   W_o[8,37] := -0.1157986;
   W_o[8,38] := 0.2580299;
   W_o[8,39] := 0.220136;
   W_o[9,0] := -0.3132641;
   W_o[9,1] := -0.06183321;
   W_o[9,2] := -0.1190897;
   W_o[9,3] := -0.1472712;
   W_o[9,4] := -0.2051323;
   W_o[9,5] := -0.619219;
   W_o[9,6] := 0.1387524;
   W_o[9,7] := -0.3166307;
   W_o[9,8] := -0.9589977;
   W_o[9,9] := 0.0739672;
   W_o[9,10] := -0.3332131;
   W_o[9,11] := 0.07539017;
   W_o[9,12] := 0.04058671;
   W_o[9,13] := -0.03272064;
   W_o[9,14] := 0.00082348;
   W_o[9,15] := 0.03252422;
   W_o[9,16] := -0.187089;
   W_o[9,17] := 0.03206202;
   W_o[9,18] := -0.1109974;
   W_o[9,19] := -0.2095204;
   W_o[9,20] := -0.5135113;
   W_o[9,21] := 0.1920649;
   W_o[9,22] := -0.01424127;
   W_o[9,23] := -0.00173319;
   W_o[9,24] := -0.08532184;
   W_o[9,25] := -0.2821319;
   W_o[9,26] := -0.03178848;
   W_o[9,27] := -0.0577799;
   W_o[9,28] := 0.2315015;
   W_o[9,29] := 0.07085361;
   W_o[9,30] := 0.1951047;
   W_o[9,31] := 0.08876722;
   W_o[9,32] := 0.1402373;
   W_o[9,33] := 0.2821989;
   W_o[9,34] := 0.1606525;
   W_o[9,35] := -0.1928923;
   W_o[9,36] := 0.01568728;
   W_o[9,37] := -0.1860046;
   W_o[9,38] := 0.09268271;
   W_o[9,39] := -0.01587286;
   W_o[10,0] := -0.02192705;
   W_o[10,1] := 0.2329542;
   W_o[10,2] := -0.00188665;
   W_o[10,3] := 0.143792;
   W_o[10,4] := 0.2532279;
   W_o[10,5] := 0.4542165;
   W_o[10,6] := 0.3260326;
   W_o[10,7] := 0.1298785;
   W_o[10,8] := -0.03717055;
   W_o[10,9] := 0.06002445;
   W_o[10,10] := -0.01521991;
   W_o[10,11] := -0.3110218;
   W_o[10,12] := -0.2009706;
   W_o[10,13] := 0.05733368;
   W_o[10,14] := -0.3404011;
   W_o[10,15] := -0.4737233;
   W_o[10,16] := 0.03586001;
   W_o[10,17] := 0.122371;
   W_o[10,18] := 0.3001329;
   W_o[10,19] := -0.05952299;
   W_o[10,20] := -0.1222852;
   W_o[10,21] := 0.1644575;
   W_o[10,22] := 0.350365;
   W_o[10,23] := -0.3212706;
   W_o[10,24] := 1.075127;
   W_o[10,25] := 1.031375;
   W_o[10,26] := -0.0865766;
   W_o[10,27] := -0.3474564;
   W_o[10,28] := 0.09863426;
   W_o[10,29] := -0.2132783;
   W_o[10,30] := 0.3851247;
   W_o[10,31] := 0.1182251;
   W_o[10,32] := 0.3440039;
   W_o[10,33] := 0.3899197;
   W_o[10,34] := 0.7392653;
   W_o[10,35] := 0.2004149;
   W_o[10,36] := -0.05608039;
   W_o[10,37] := 0.2275992;
   W_o[10,38] := -0.04267087;
   W_o[10,39] := 0.2836826;
   W_o[11,0] := -0.1809653;
   W_o[11,1] := 0.1015071;
   W_o[11,2] := -0.1359787;
   W_o[11,3] := -0.339222;
   W_o[11,4] := 0.01738593;
   W_o[11,5] := 0.00192241;
   W_o[11,6] := -0.02194121;
   W_o[11,7] := -0.1547077;
   W_o[11,8] := 0.06660517;
   W_o[11,9] := -0.1348383;
   W_o[11,10] := -0.134767;
   W_o[11,11] := -0.1782693;
   W_o[11,12] := 0.1472701;
   W_o[11,13] := -0.2786617;
   W_o[11,14] := 0.09056337;
   W_o[11,15] := -0.07600223;
   W_o[11,16] := 0.0426885;
   W_o[11,17] := 0.1939706;
   W_o[11,18] := 0.06352299;
   W_o[11,19] := -0.3184692;
   W_o[11,20] := -0.08175273;
   W_o[11,21] := 0.156256;
   W_o[11,22] := -0.1318633;
   W_o[11,23] := -0.4227056;
   W_o[11,24] := 0.03163491;
   W_o[11,25] := 0.3073466;
   W_o[11,26] := 0.1847536;
   W_o[11,27] := -0.1969137;
   W_o[11,28] := 0.1285785;
   W_o[11,29] := 0.02137278;
   W_o[11,30] := -0.08936202;
   W_o[11,31] := 0.2781714;
   W_o[11,32] := -0.09503862;
   W_o[11,33] := -0.1658657;
   W_o[11,34] := -0.1278383;
   W_o[11,35] := -0.1624458;
   W_o[11,36] := 0.1902921;
   W_o[11,37] := 0.127865;
   W_o[11,38] := -0.07075812;
   W_o[11,39] := 0.428382;
   W_o[12,0] := -0.1219991;
   W_o[12,1] := 0.03823468;
   W_o[12,2] := 0.01577434;
   W_o[12,3] := 0.1470047;
   W_o[12,4] := 0.0760267;
   W_o[12,5] := -0.05943288;
   W_o[12,6] := 0.1218424;
   W_o[12,7] := -0.4092018;
   W_o[12,8] := -0.01477545;
   W_o[12,9] := 0.1050386;
   W_o[12,10] := -0.06524223;
   W_o[12,11] := -0.04999274;
   W_o[12,12] := 0.3521778;
   W_o[12,13] := -0.07877419;
   W_o[12,14] := 0.09900068;
   W_o[12,15] := 0.05063246;
   W_o[12,16] := 0.1021576;
   W_o[12,17] := -0.1172289;
   W_o[12,18] := 0.0756586;
   W_o[12,19] := -0.08223618;
   W_o[12,20] := -0.2851469;
   W_o[12,21] := -0.00324072;
   W_o[12,22] := 0.0636245;
   W_o[12,23] := -0.1829358;
   W_o[12,24] := -0.3075816;
   W_o[12,25] := -0.2720142;
   W_o[12,26] := 0.1688922;
   W_o[12,27] := 0.06790268;
   W_o[12,28] := 0.09229479;
   W_o[12,29] := -0.02702256;
   W_o[12,30] := 0.04384379;
   W_o[12,31] := -0.2710299;
   W_o[12,32] := -0.1930007;
   W_o[12,33] := 0.3236164;
   W_o[12,34] := 0.00694379;
   W_o[12,35] := 0.05657077;
   W_o[12,36] := -0.1271545;
   W_o[12,37] := -0.1242922;
   W_o[12,38] := 0.2896774;
   W_o[12,39] := -0.08116662;
   W_o[13,0] := 0.368947;
   W_o[13,1] := 0.1130772;
   W_o[13,2] := 0.5471025;
   W_o[13,3] := -0.3829838;
   W_o[13,4] := 0.6498483;
   W_o[13,5] := -0.2602773;
   W_o[13,6] := 0.2094651;
   W_o[13,7] := 0.02607361;
   W_o[13,8] := -0.1112638;
   W_o[13,9] := -0.06411502;
   W_o[13,10] := -0.03624791;
   W_o[13,11] := -0.04085876;
   W_o[13,12] := -0.3497492;
   W_o[13,13] := -0.1605573;
   W_o[13,14] := 0.1782783;
   W_o[13,15] := -0.04494572;
   W_o[13,16] := 0.1499656;
   W_o[13,17] := -0.1109314;
   W_o[13,18] := 0.5331051;
   W_o[13,19] := -0.4442391;
   W_o[13,20] := -0.07231531;
   W_o[13,21] := 0.3642985;
   W_o[13,22] := 0.5776525;
   W_o[13,23] := -0.1446741;
   W_o[13,24] := 1.537843;
   W_o[13,25] := 1.406464;
   W_o[13,26] := -0.1982083;
   W_o[13,27] := 0.2525975;
   W_o[13,28] := 0.1090571;
   W_o[13,29] := -0.3863609;
   W_o[13,30] := 0.3198679;
   W_o[13,31] := -0.0655776;
   W_o[13,32] := 0.1591396;
   W_o[13,33] := 0.3302372;
   W_o[13,34] := 0.8010866;
   W_o[13,35] := 0.00219575;
   W_o[13,36] := 0.3194016;
   W_o[13,37] := 0.3292364;
   W_o[13,38] := 0.2895371;
   W_o[13,39] := 0.1438104;
   W_o[14,0] := -0.06043304;
   W_o[14,1] := 0.1463838;
   W_o[14,2] := 0.1813115;
   W_o[14,3] := -0.4461174;
   W_o[14,4] := -0.08022243;
   W_o[14,5] := 0.1215249;
   W_o[14,6] := -0.09096271;
   W_o[14,7] := -0.08817829;
   W_o[14,8] := -0.4104892;
   W_o[14,9] := 0.00550563;
   W_o[14,10] := 0.02338252;
   W_o[14,11] := 0.03576816;
   W_o[14,12] := 0.09025624;
   W_o[14,13] := -0.165952;
   W_o[14,14] := -0.1859627;
   W_o[14,15] := -0.09394215;
   W_o[14,16] := -0.06208068;
   W_o[14,17] := -0.00717838;
   W_o[14,18] := 0.1996924;
   W_o[14,19] := 0.01073706;
   W_o[14,20] := -0.1823136;
   W_o[14,21] := 0.01420894;
   W_o[14,22] := -0.1017454;
   W_o[14,23] := -0.4975724;
   W_o[14,24] := -0.4672968;
   W_o[14,25] := -0.2924049;
   W_o[14,26] := -0.190528;
   W_o[14,27] := -0.1670942;
   W_o[14,28] := -0.01935058;
   W_o[14,29] := -0.1424983;
   W_o[14,30] := -0.1588129;
   W_o[14,31] := 0.2039351;
   W_o[14,32] := -0.06176985;
   W_o[14,33] := 0.1746421;
   W_o[14,34] := 0.2394749;
   W_o[14,35] := -0.1960727;
   W_o[14,36] := 0.05518134;
   W_o[14,37] := 0.09389904;
   W_o[14,38] := 0.08116579;
   W_o[14,39] := 0.1385406;
   W_o[15,0] := -0.2035415;
   W_o[15,1] := 0.2229884;
   W_o[15,2] := -0.7284631;
   W_o[15,3] := 0.1279051;
   W_o[15,4] := -0.000869;
   W_o[15,5] := 0.5366808;
   W_o[15,6] := -0.01224643;
   W_o[15,7] := 0.1336179;
   W_o[15,8] := -0.3520414;
   W_o[15,9] := -0.00480295;
   W_o[15,10] := 0.1333943;
   W_o[15,11] := 0.05102095;
   W_o[15,12] := -0.05708028;
   W_o[15,13] := -0.06014942;
   W_o[15,14] := 0.01049514;
   W_o[15,15] := -0.09353844;
   W_o[15,16] := 0.07731096;
   W_o[15,17] := 0.01013883;
   W_o[15,18] := 0.07310723;
   W_o[15,19] := -0.8692668;
   W_o[15,20] := -0.2155429;
   W_o[15,21] := 0.09906635;
   W_o[15,22] := -0.0306251;
   W_o[15,23] := 0.3455428;
   W_o[15,24] := -0.1861183;
   W_o[15,25] := -0.2109679;
   W_o[15,26] := -0.05899647;
   W_o[15,27] := 0.01260784;
   W_o[15,28] := 0.04030582;
   W_o[15,29] := 0.1423471;
   W_o[15,30] := 0.2868683;
   W_o[15,31] := 0.1026989;
   W_o[15,32] := 0.2412259;
   W_o[15,33] := -0.04419544;
   W_o[15,34] := 0.1289678;
   W_o[15,35] := -0.2943439;
   W_o[15,36] := -0.00652304;
   W_o[15,37] := -0.03412445;
   W_o[15,38] := 0.4802624;
   W_o[15,39] := 0.2227584;
   R_i[0,0] := -0.01601154;
   R_i[0,1] := -0.4505664;
   R_i[0,2] := 0.3115061;
   R_i[0,3] := 0.7538006;
   R_i[0,4] := -0.1402078;
   R_i[0,5] := -0.04954997;
   R_i[0,6] := -0.08327835;
   R_i[0,7] := 0.3733349;
   R_i[0,8] := 0.6963265;
   R_i[0,9] := 0.2863626;
   R_i[0,10] := 0.7997712;
   R_i[0,11] := -0.7498176;
   R_i[0,12] := -0.6526057;
   R_i[0,13] := 0.1387625;
   R_i[0,14] := 0.08631746;
   R_i[0,15] := 0.05898035;
   R_i[1,0] := -0.401232;
   R_i[1,1] := 0.7335209;
   R_i[1,2] := -0.09579885;
   R_i[1,3] := 0.02985846;
   R_i[1,4] := -0.3186485;
   R_i[1,5] := -0.2394537;
   R_i[1,6] := 0.5418519;
   R_i[1,7] := -0.2710277;
   R_i[1,8] := 0.00622073;
   R_i[1,9] := 0.09155256;
   R_i[1,10] := 0.1461604;
   R_i[1,11] := -0.0016893;
   R_i[1,12] := 0.2237979;
   R_i[1,13] := 0.1673195;
   R_i[1,14] := -0.07847317;
   R_i[1,15] := -0.07302959;
   R_i[2,0] := 0.2143267;
   R_i[2,1] := -0.5247285;
   R_i[2,2] := 0.3322655;
   R_i[2,3] := 0.2965375;
   R_i[2,4] := 0.1318167;
   R_i[2,5] := 0.1446274;
   R_i[2,6] := -0.130442;
   R_i[2,7] := -0.1195364;
   R_i[2,8] := -0.3126507;
   R_i[2,9] := -0.240243;
   R_i[2,10] := 0.08897854;
   R_i[2,11] := -0.3383393;
   R_i[2,12] := -0.1979901;
   R_i[2,13] := 0.07993159;
   R_i[2,14] := -0.1129293;
   R_i[2,15] := -0.07898453;
   R_i[3,0] := 0.2161791;
   R_i[3,1] := 0.14047;
   R_i[3,2] := -0.339711;
   R_i[3,3] := -0.8781343;
   R_i[3,4] := 0.1890773;
   R_i[3,5] := -0.08525109;
   R_i[3,6] := 0.00524858;
   R_i[3,7] := 0.6169428;
   R_i[3,8] := -0.02290213;
   R_i[3,9] := -0.1232494;
   R_i[3,10] := 0.1836437;
   R_i[3,11] := -0.0097614;
   R_i[3,12] := -0.00912099;
   R_i[3,13] := 0.08642489;
   R_i[3,14] := -0.1198076;
   R_i[3,15] := -0.1218542;
   R_i[4,0] := -0.1688442;
   R_i[4,1] := -0.01549527;
   R_i[4,2] := -0.09087992;
   R_i[4,3] := 0.2035424;
   R_i[4,4] := 0.03523245;
   R_i[4,5] := -0.7966576;
   R_i[4,6] := 0.01135984;
   R_i[4,7] := 0.1643567;
   R_i[4,8] := 0.2464019;
   R_i[4,9] := 0.348982;
   R_i[4,10] := 0.1028246;
   R_i[4,11] := 0.00752686;
   R_i[4,12] := 0.04740289;
   R_i[4,13] := 0.6564606;
   R_i[4,14] := 0.3415406;
   R_i[4,15] := -0.1820581;
   R_i[5,0] := 0.14134;
   R_i[5,1] := -0.5241947;
   R_i[5,2] := 0.2979371;
   R_i[5,3] := 0.5492764;
   R_i[5,4] := -0.5426098;
   R_i[5,5] := -0.5120263;
   R_i[5,6] := -0.6021063;
   R_i[5,7] := -0.5658756;
   R_i[5,8] := 0.2832164;
   R_i[5,9] := 0.2791682;
   R_i[5,10] := 0.0495842;
   R_i[5,11] := -0.4578474;
   R_i[5,12] := -0.6485385;
   R_i[5,13] := 0.06905902;
   R_i[5,14] := -0.4043413;
   R_i[5,15] := -0.3203804;
   R_i[6,0] := -0.1409825;
   R_i[6,1] := -0.5848475;
   R_i[6,2] := 0.1453531;
   R_i[6,3] := 0.07121052;
   R_i[6,4] := -0.3604121;
   R_i[6,5] := -0.397943;
   R_i[6,6] := -1.122013;
   R_i[6,7] := -0.1309183;
   R_i[6,8] := -0.191392;
   R_i[6,9] := 0.02611434;
   R_i[6,10] := -0.2210553;
   R_i[6,11] := 0.03291342;
   R_i[6,12] := -0.3278158;
   R_i[6,13] := 0.3461519;
   R_i[6,14] := 0.2672345;
   R_i[6,15] := 0.1619738;
   R_i[7,0] := -0.1475523;
   R_i[7,1] := -0.6828271;
   R_i[7,2] := -0.2710959;
   R_i[7,3] := 0.3215815;
   R_i[7,4] := 0.03019373;
   R_i[7,5] := 0.1696624;
   R_i[7,6] := 0.1198417;
   R_i[7,7] := -0.1019654;
   R_i[7,8] := 0.5909069;
   R_i[7,9] := -0.3902815;
   R_i[7,10] := 0.2400998;
   R_i[7,11] := -0.3905518;
   R_i[7,12] := -0.3868088;
   R_i[7,13] := -0.1764367;
   R_i[7,14] := 0.2387517;
   R_i[7,15] := -0.1071883;
   R_i[8,0] := -0.23345;
   R_i[8,1] := -0.3877599;
   R_i[8,2] := -0.3317247;
   R_i[8,3] := 0.1490105;
   R_i[8,4] := 0.07190004;
   R_i[8,5] := -0.05165868;
   R_i[8,6] := 0.4919274;
   R_i[8,7] := 0.6358661;
   R_i[8,8] := -0.1297378;
   R_i[8,9] := -0.3915481;
   R_i[8,10] := 0.01818666;
   R_i[8,11] := -0.3103262;
   R_i[8,12] := -0.2901289;
   R_i[8,13] := -0.01039465;
   R_i[8,14] := 0.194509;
   R_i[8,15] := -0.2007908;
   R_i[9,0] := -0.2780712;
   R_i[9,1] := 0.00795646;
   R_i[9,2] := 0.1596926;
   R_i[9,3] := -0.09819215;
   R_i[9,4] := 0.00536336;
   R_i[9,5] := -0.01222592;
   R_i[9,6] := 0.05426886;
   R_i[9,7] := -0.2209529;
   R_i[9,8] := 0.1505673;
   R_i[9,9] := -0.2607254;
   R_i[9,10] := 0.3316929;
   R_i[9,11] := 0.1011708;
   R_i[9,12] := -0.2139317;
   R_i[9,13] := 0.4217584;
   R_i[9,14] := 0.01216281;
   R_i[9,15] := -0.0816205;
   R_i[10,0] := 0.126458;
   R_i[10,1] := 0.02421534;
   R_i[10,2] := -0.2489259;
   R_i[10,3] := 0.09164374;
   R_i[10,4] := -0.4294859;
   R_i[10,5] := -0.0543494;
   R_i[10,6] := 0.5646753;
   R_i[10,7] := 0.331787;
   R_i[10,8] := 0.2602156;
   R_i[10,9] := -0.3929808;
   R_i[10,10] := -0.395796;
   R_i[10,11] := -0.00741246;
   R_i[10,12] := -0.3358352;
   R_i[10,13] := -0.0185852;
   R_i[10,14] := 0.4410301;
   R_i[10,15] := -0.09651927;
   R_i[11,0] := 0.09693456;
   R_i[11,1] := -0.3512501;
   R_i[11,2] := -0.02015482;
   R_i[11,3] := 0.3572097;
   R_i[11,4] := -0.1196542;
   R_i[11,5] := 0.1445999;
   R_i[11,6] := -0.1906793;
   R_i[11,7] := 0.08080416;
   R_i[11,8] := 0.1779785;
   R_i[11,9] := -0.1425034;
   R_i[11,10] := -0.3862794;
   R_i[11,11] := 0.4956163;
   R_i[11,12] := -0.1790929;
   R_i[11,13] := 0.2083636;
   R_i[11,14] := 0.4006914;
   R_i[11,15] := 0.3896022;
   R_i[12,0] := 0.3400891;
   R_i[12,1] := -0.1727159;
   R_i[12,2] := -0.3076965;
   R_i[12,3] := -0.2823079;
   R_i[12,4] := 0.0525449;
   R_i[12,5] := 0.07448359;
   R_i[12,6] := -0.00981909;
   R_i[12,7] := 0.1008154;
   R_i[12,8] := 0.3009783;
   R_i[12,9] := 0.2912007;
   R_i[12,10] := 0.1271894;
   R_i[12,11] := -0.06783659;
   R_i[12,12] := 0.4455962;
   R_i[12,13] := -0.3242948;
   R_i[12,14] := -0.183432;
   R_i[12,15] := -0.1089303;
   R_i[13,0] := -0.2894851;
   R_i[13,1] := -0.1664966;
   R_i[13,2] := 0.04430598;
   R_i[13,3] := 0.1107857;
   R_i[13,4] := -0.5688026;
   R_i[13,5] := -0.07979194;
   R_i[13,6] := 0.1527517;
   R_i[13,7] := 0.1273375;
   R_i[13,8] := 0.3621153;
   R_i[13,9] := 0.3043333;
   R_i[13,10] := -0.1798581;
   R_i[13,11] := -0.237729;
   R_i[13,12] := 0.1235583;
   R_i[13,13] := 0.5035439;
   R_i[13,14] := 0.108624;
   R_i[13,15] := -0.02580172;
   R_i[14,0] := 0.04543614;
   R_i[14,1] := -0.4043088;
   R_i[14,2] := 0.1209751;
   R_i[14,3] := 0.4883763;
   R_i[14,4] := 0.00980398;
   R_i[14,5] := 0.03799421;
   R_i[14,6] := 0.3278515;
   R_i[14,7] := 0.0660439;
   R_i[14,8] := 0.172085;
   R_i[14,9] := -0.3707425;
   R_i[14,10] := -0.1385914;
   R_i[14,11] := 0.2718971;
   R_i[14,12] := -0.1328888;
   R_i[14,13] := 0.2701875;
   R_i[14,14] := 1.386678;
   R_i[14,15] := 0.05095792;
   R_i[15,0] := 0.1214196;
   R_i[15,1] := -0.03100028;
   R_i[15,2] := 0.2684634;
   R_i[15,3] := 0.2103243;
   R_i[15,4] := -0.1190422;
   R_i[15,5] := 0.09452529;
   R_i[15,6] := 0.3082354;
   R_i[15,7] := -3.856E-05;
   R_i[15,8] := 0.2727255;
   R_i[15,9] := 0.05441154;
   R_i[15,10] := -0.1230815;
   R_i[15,11] := -0.4781843;
   R_i[15,12] := -0.2143165;
   R_i[15,13] := -0.2471516;
   R_i[15,14] := 0.2087188;
   R_i[15,15] := 0.02325043;
   R_f[0,0] := -0.03493118;
   R_f[0,1] := -0.3783333;
   R_f[0,2] := 0.03728793;
   R_f[0,3] := 0.1427855;
   R_f[0,4] := -0.1200396;
   R_f[0,5] := -0.06856227;
   R_f[0,6] := 0.07930882;
   R_f[0,7] := 0.2776607;
   R_f[0,8] := 0.07494716;
   R_f[0,9] := 0.1461581;
   R_f[0,10] := -0.07652009;
   R_f[0,11] := -0.09052465;
   R_f[0,12] := -0.1157662;
   R_f[0,13] := 0.04987612;
   R_f[0,14] := 0.06529343;
   R_f[0,15] := 0.00263772;
   R_f[1,0] := -0.4377774;
   R_f[1,1] := 0.7251403;
   R_f[1,2] := -0.3877139;
   R_f[1,3] := -0.0144369;
   R_f[1,4] := -0.00149874;
   R_f[1,5] := -0.3447672;
   R_f[1,6] := 0.2917376;
   R_f[1,7] := 0.09541123;
   R_f[1,8] := 0.3457976;
   R_f[1,9] := 0.6298571;
   R_f[1,10] := 0.05302448;
   R_f[1,11] := 0.2072578;
   R_f[1,12] := -0.04234733;
   R_f[1,13] := 0.3336825;
   R_f[1,14] := 0.1307107;
   R_f[1,15] := 0.1257179;
   R_f[2,0] := 0.3310767;
   R_f[2,1] := -0.3810703;
   R_f[2,2] := 0.1153975;
   R_f[2,3] := 0.3476575;
   R_f[2,4] := -0.2480675;
   R_f[2,5] := 0.1239669;
   R_f[2,6] := -0.0001569;
   R_f[2,7] := -0.03111286;
   R_f[2,8] := -0.4061953;
   R_f[2,9] := -0.1027613;
   R_f[2,10] := -0.01848604;
   R_f[2,11] := -0.3815011;
   R_f[2,12] := 0.07561549;
   R_f[2,13] := -0.3294232;
   R_f[2,14] := -0.04146929;
   R_f[2,15] := 0.1021808;
   R_f[3,0] := -0.9564785;
   R_f[3,1] := 0.3263851;
   R_f[3,2] := -0.1824219;
   R_f[3,3] := -0.2994925;
   R_f[3,4] := 0.1714023;
   R_f[3,5] := -0.2092119;
   R_f[3,6] := -0.1032977;
   R_f[3,7] := -0.1582146;
   R_f[3,8] := 0.1507048;
   R_f[3,9] := 0.337986;
   R_f[3,10] := -0.2794919;
   R_f[3,11] := 0.08474356;
   R_f[3,12] := 0.2481105;
   R_f[3,13] := 0.09939278;
   R_f[3,14] := -0.2410131;
   R_f[3,15] := -0.1935376;
   R_f[4,0] := -0.234988;
   R_f[4,1] := -0.4074499;
   R_f[4,2] := 0.2635157;
   R_f[4,3] := -0.2668453;
   R_f[4,4] := -0.09082807;
   R_f[4,5] := -0.08405253;
   R_f[4,6] := 0.08696185;
   R_f[4,7] := 0.1112983;
   R_f[4,8] := 0.1638763;
   R_f[4,9] := -0.1186807;
   R_f[4,10] := 0.3262174;
   R_f[4,11] := -0.1426349;
   R_f[4,12] := 0.1308399;
   R_f[4,13] := 0.1795556;
   R_f[4,14] := 0.1659483;
   R_f[4,15] := 0.1235942;
   R_f[5,0] := 0.3548082;
   R_f[5,1] := -0.1270981;
   R_f[5,2] := 0.2426847;
   R_f[5,3] := 0.0801195;
   R_f[5,4] := 0.2115624;
   R_f[5,5] := 0.2757975;
   R_f[5,6] := 0.2001711;
   R_f[5,7] := 0.01883883;
   R_f[5,8] := -0.3942798;
   R_f[5,9] := -0.3586779;
   R_f[5,10] := 0.06389395;
   R_f[5,11] := -0.1110686;
   R_f[5,12] := 0.1175703;
   R_f[5,13] := -0.0187532;
   R_f[5,14] := 0.01303833;
   R_f[5,15] := -0.0669001;
   R_f[6,0] := -0.5004723;
   R_f[6,1] := -0.07684148;
   R_f[6,2] := 0.1981799;
   R_f[6,3] := 0.0597102;
   R_f[6,4] := -0.04680483;
   R_f[6,5] := 0.317703;
   R_f[6,6] := 0.1253361;
   R_f[6,7] := 0.1381588;
   R_f[6,8] := 0.02148284;
   R_f[6,9] := -0.0610669;
   R_f[6,10] := 0.1336211;
   R_f[6,11] := 0.2163607;
   R_f[6,12] := -0.09828766;
   R_f[6,13] := 0.2164403;
   R_f[6,14] := 0.2033899;
   R_f[6,15] := 0.1417818;
   R_f[7,0] := 0.2612512;
   R_f[7,1] := -0.03714739;
   R_f[7,2] := 0.08117681;
   R_f[7,3] := 0.20745;
   R_f[7,4] := -0.320446;
   R_f[7,5] := 0.4126448;
   R_f[7,6] := 0.616157;
   R_f[7,7] := -0.1764756;
   R_f[7,8] := -0.1566713;
   R_f[7,9] := -0.02732511;
   R_f[7,10] := -0.4989151;
   R_f[7,11] := 0.00061774;
   R_f[7,12] := -0.02982556;
   R_f[7,13] := 0.03914607;
   R_f[7,14] := 0.2035217;
   R_f[7,15] := 0.01521025;
   R_f[8,0] := -0.00262567;
   R_f[8,1] := -0.1957263;
   R_f[8,2] := -0.0133352;
   R_f[8,3] := 0.1326498;
   R_f[8,4] := -0.06475109;
   R_f[8,5] := 0.2750055;
   R_f[8,6] := 0.2935895;
   R_f[8,7] := 0.1078199;
   R_f[8,8] := -0.5541819;
   R_f[8,9] := -0.03762578;
   R_f[8,10] := -0.2519385;
   R_f[8,11] := 0.277219;
   R_f[8,12] := -0.1539617;
   R_f[8,13] := -0.02145483;
   R_f[8,14] := 0.2416782;
   R_f[8,15] := 0.06824671;
   R_f[9,0] := 0.2504059;
   R_f[9,1] := -0.3383861;
   R_f[9,2] := 0.0674123;
   R_f[9,3] := 0.2097046;
   R_f[9,4] := -0.0898691;
   R_f[9,5] := -0.2091327;
   R_f[9,6] := 0.3162811;
   R_f[9,7] := 0.265341;
   R_f[9,8] := 0.02326944;
   R_f[9,9] := -0.8053678;
   R_f[9,10] := -0.2416072;
   R_f[9,11] := -0.03336972;
   R_f[9,12] := -0.3634549;
   R_f[9,13] := 0.01661946;
   R_f[9,14] := -0.117901;
   R_f[9,15] := 0.1400468;
   R_f[10,0] := 0.2025216;
   R_f[10,1] := -0.3309455;
   R_f[10,2] := 0.2834905;
   R_f[10,3] := 0.2098317;
   R_f[10,4] := -0.3916658;
   R_f[10,5] := 0.1489443;
   R_f[10,6] := 0.05038162;
   R_f[10,7] := 0.1421797;
   R_f[10,8] := -0.2475107;
   R_f[10,9] := 0.04759743;
   R_f[10,10] := -0.1642638;
   R_f[10,11] := -0.1621708;
   R_f[10,12] := -0.1235068;
   R_f[10,13] := 0.08995254;
   R_f[10,14] := -0.01327613;
   R_f[10,15] := 0.2285491;
   R_f[11,0] := 0.1601221;
   R_f[11,1] := 0.2628818;
   R_f[11,2] := 0.2190603;
   R_f[11,3] := -0.04701964;
   R_f[11,4] := -0.1388493;
   R_f[11,5] := 0.08709867;
   R_f[11,6] := -0.07009537;
   R_f[11,7] := -0.1695109;
   R_f[11,8] := 0.02868164;
   R_f[11,9] := -0.0112115;
   R_f[11,10] := 0.07267684;
   R_f[11,11] := -0.1989551;
   R_f[11,12] := 0.3613658;
   R_f[11,13] := -0.05935945;
   R_f[11,14] := 0.0822355;
   R_f[11,15] := 0.373795;
   R_f[12,0] := -0.2599636;
   R_f[12,1] := -0.4840415;
   R_f[12,2] := -0.3295081;
   R_f[12,3] := 0.1110019;
   R_f[12,4] := -0.2677098;
   R_f[12,5] := -0.1735305;
   R_f[12,6] := 0.1697096;
   R_f[12,7] := -0.3476382;
   R_f[12,8] := 0.517248;
   R_f[12,9] := -0.2285556;
   R_f[12,10] := 0.86062;
   R_f[12,11] := 0.06095523;
   R_f[12,12] := -0.1267713;
   R_f[12,13] := 0.2335584;
   R_f[12,14] := 0.2402046;
   R_f[12,15] := -0.2279788;
   R_f[13,0] := 0.02567713;
   R_f[13,1] := -0.3151536;
   R_f[13,2] := -0.1262183;
   R_f[13,3] := 0.1836853;
   R_f[13,4] := -0.03905401;
   R_f[13,5] := 0.7135632;
   R_f[13,6] := 0.08130559;
   R_f[13,7] := 0.01576971;
   R_f[13,8] := -0.2050417;
   R_f[13,9] := 0.07079811;
   R_f[13,10] := -0.1090281;
   R_f[13,11] := 0.1574726;
   R_f[13,12] := -0.3404612;
   R_f[13,13] := 0.1042019;
   R_f[13,14] := -0.05406023;
   R_f[13,15] := 0.2302613;
   R_f[14,0] := 0.05553682;
   R_f[14,1] := 0.03039004;
   R_f[14,2] := -0.3977577;
   R_f[14,3] := 0.1773666;
   R_f[14,4] := -0.1401487;
   R_f[14,5] := 0.1813615;
   R_f[14,6] := 0.08784663;
   R_f[14,7] := -0.00406716;
   R_f[14,8] := 0.2937247;
   R_f[14,9] := -0.2185726;
   R_f[14,10] := 0.3286898;
   R_f[14,11] := 0.5202897;
   R_f[14,12] := 0.2797473;
   R_f[14,13] := -0.109547;
   R_f[14,14] := 1.174732;
   R_f[14,15] := 0.2927172;
   R_f[15,0] := 0.3542146;
   R_f[15,1] := -0.6242056;
   R_f[15,2] := 0.2294325;
   R_f[15,3] := 0.2983122;
   R_f[15,4] := -0.2018091;
   R_f[15,5] := 0.3988208;
   R_f[15,6] := 0.2762798;
   R_f[15,7] := 0.3846879;
   R_f[15,8] := 0.04349254;
   R_f[15,9] := -0.1081066;
   R_f[15,10] := -0.3734537;
   R_f[15,11] := -0.1098458;
   R_f[15,12] := 0.3364737;
   R_f[15,13] := 0.3455147;
   R_f[15,14] := 0.02944022;
   R_f[15,15] := 0.02307001;
   R_g[0,0] := -1.251124;
   R_g[0,1] := -0.2188334;
   R_g[0,2] := 0.1101293;
   R_g[0,3] := 0.2501267;
   R_g[0,4] := -0.1040586;
   R_g[0,5] := 0.1389121;
   R_g[0,6] := 0.1024126;
   R_g[0,7] := 0.2224759;
   R_g[0,8] := 0.06886309;
   R_g[0,9] := -0.05504098;
   R_g[0,10] := 0.1316268;
   R_g[0,11] := -0.09226879;
   R_g[0,12] := 0.03665201;
   R_g[0,13] := 0.01448225;
   R_g[0,14] := 0.08514914;
   R_g[0,15] := 0.1034982;
   R_g[1,0] := -0.01289242;
   R_g[1,1] := -0.7693796;
   R_g[1,2] := -0.00765862;
   R_g[1,3] := -0.02182954;
   R_g[1,4] := -0.0062479;
   R_g[1,5] := -0.09856889;
   R_g[1,6] := -0.00179921;
   R_g[1,7] := -0.1597593;
   R_g[1,8] := 0.1441042;
   R_g[1,9] := -0.136594;
   R_g[1,10] := -0.1046183;
   R_g[1,11] := 0.1787898;
   R_g[1,12] := 0.1371266;
   R_g[1,13] := 0.1039945;
   R_g[1,14] := 0.2064357;
   R_g[1,15] := 0.05955669;
   R_g[2,0] := -0.00450423;
   R_g[2,1] := 0.2783746;
   R_g[2,2] := -1.652401;
   R_g[2,3] := -0.08348246;
   R_g[2,4] := 0.00295603;
   R_g[2,5] := -0.1220379;
   R_g[2,6] := -0.01780931;
   R_g[2,7] := 0.08614038;
   R_g[2,8] := -0.05562058;
   R_g[2,9] := 0.1005678;
   R_g[2,10] := 0.03247114;
   R_g[2,11] := -0.1122308;
   R_g[2,12] := -0.1009854;
   R_g[2,13] := 0.01667355;
   R_g[2,14] := -0.2604633;
   R_g[2,15] := -0.262483;
   R_g[3,0] := -0.03127015;
   R_g[3,1] := 0.2364704;
   R_g[3,2] := -0.2546491;
   R_g[3,3] := -0.9946523;
   R_g[3,4] := -0.00474326;
   R_g[3,5] := 0.0225782;
   R_g[3,6] := -0.1201107;
   R_g[3,7] := -0.3624461;
   R_g[3,8] := 0.1697178;
   R_g[3,9] := 0.1855698;
   R_g[3,10] := 0.1265972;
   R_g[3,11] := -0.07901487;
   R_g[3,12] := -0.08990744;
   R_g[3,13] := 0.1421835;
   R_g[3,14] := -0.143879;
   R_g[3,15] := -0.2938069;
   R_g[4,0] := 0.07746305;
   R_g[4,1] := 0.05525218;
   R_g[4,2] := 0.1861004;
   R_g[4,3] := 0.1101569;
   R_g[4,4] := -1.795932;
   R_g[4,5] := -0.03749003;
   R_g[4,6] := 0.01035422;
   R_g[4,7] := 0.1005974;
   R_g[4,8] := 0.2383393;
   R_g[4,9] := -0.04896057;
   R_g[4,10] := -0.1035081;
   R_g[4,11] := 0.0563738;
   R_g[4,12] := -0.2545002;
   R_g[4,13] := -0.08886177;
   R_g[4,14] := -0.115833;
   R_g[4,15] := 0.4366852;
   R_g[5,0] := -0.1500607;
   R_g[5,1] := 0.1485784;
   R_g[5,2] := 0.09219331;
   R_g[5,3] := 0.2430712;
   R_g[5,4] := 0.02014972;
   R_g[5,5] := -1.739048;
   R_g[5,6] := -0.06327479;
   R_g[5,7] := 0.09475522;
   R_g[5,8] := -0.0571667;
   R_g[5,9] := 0.00648821;
   R_g[5,10] := -0.08605717;
   R_g[5,11] := 0.04396249;
   R_g[5,12] := 0.1986526;
   R_g[5,13] := 0.2101544;
   R_g[5,14] := -0.04510098;
   R_g[5,15] := -0.05707484;
   R_g[6,0] := 0.05463404;
   R_g[6,1] := -0.2467168;
   R_g[6,2] := 0.1494595;
   R_g[6,3] := 0.2778161;
   R_g[6,4] := 0.05857803;
   R_g[6,5] := -0.09827307;
   R_g[6,6] := -1.369555;
   R_g[6,7] := 0.03997089;
   R_g[6,8] := 0.1069783;
   R_g[6,9] := -0.152829;
   R_g[6,10] := -0.1145824;
   R_g[6,11] := 0.2323128;
   R_g[6,12] := 0.06463466;
   R_g[6,13] := -0.04114177;
   R_g[6,14] := 0.01473683;
   R_g[6,15] := 0.09800901;
   R_g[7,0] := 0.03089882;
   R_g[7,1] := -0.1286617;
   R_g[7,2] := -0.1448888;
   R_g[7,3] := 0.08099888;
   R_g[7,4] := -0.01760847;
   R_g[7,5] := 0.123238;
   R_g[7,6] := 0.01051104;
   R_g[7,7] := -1.431484;
   R_g[7,8] := 0.05538348;
   R_g[7,9] := 0.08765257;
   R_g[7,10] := 0.04525751;
   R_g[7,11] := -0.08530193;
   R_g[7,12] := 0.06940229;
   R_g[7,13] := 0.2047146;
   R_g[7,14] := 0.1114375;
   R_g[7,15] := -0.01617558;
   R_g[8,0] := 0.00375073;
   R_g[8,1] := 0.05561948;
   R_g[8,2] := 0.07504495;
   R_g[8,3] := 0.1384679;
   R_g[8,4] := 0.01292397;
   R_g[8,5] := -0.1276252;
   R_g[8,6] := 0.00967023;
   R_g[8,7] := -0.02755805;
   R_g[8,8] := -1.648121;
   R_g[8,9] := 0.1276399;
   R_g[8,10] := 0.1534631;
   R_g[8,11] := -0.01111799;
   R_g[8,12] := 0.1786743;
   R_g[8,13] := -0.1449942;
   R_g[8,14] := -0.04605825;
   R_g[8,15] := 0.04006226;
   R_g[9,0] := 0.07299295;
   R_g[9,1] := -0.1971753;
   R_g[9,2] := -0.09354591;
   R_g[9,3] := 0.114232;
   R_g[9,4] := 0.1877067;
   R_g[9,5] := -0.1877008;
   R_g[9,6] := 0.1763708;
   R_g[9,7] := -0.00016326;
   R_g[9,8] := 0.05343577;
   R_g[9,9] := -1.985819;
   R_g[9,10] := -0.07635771;
   R_g[9,11] := 0.00779606;
   R_g[9,12] := -0.2143648;
   R_g[9,13] := 0.1459147;
   R_g[9,14] := 0.07554781;
   R_g[9,15] := -0.05975449;
   R_g[10,0] := -0.2548342;
   R_g[10,1] := 0.06535473;
   R_g[10,2] := -0.1516876;
   R_g[10,3] := -0.136762;
   R_g[10,4] := 0.1371599;
   R_g[10,5] := -0.04971113;
   R_g[10,6] := -0.04342166;
   R_g[10,7] := 0.1320384;
   R_g[10,8] := -0.05174213;
   R_g[10,9] := 0.172242;
   R_g[10,10] := -1.545853;
   R_g[10,11] := 0.08824725;
   R_g[10,12] := 0.543172;
   R_g[10,13] := -0.00582574;
   R_g[10,14] := -0.1842785;
   R_g[10,15] := -0.08446352;
   R_g[11,0] := -0.01310127;
   R_g[11,1] := 0.354282;
   R_g[11,2] := -0.2256483;
   R_g[11,3] := -0.4770394;
   R_g[11,4] := 0.02761533;
   R_g[11,5] := -0.02962572;
   R_g[11,6] := 0.06179708;
   R_g[11,7] := -0.0153362;
   R_g[11,8] := 0.04956101;
   R_g[11,9] := 0.1562686;
   R_g[11,10] := -0.1213244;
   R_g[11,11] := -0.9070006;
   R_g[11,12] := 0.2075333;
   R_g[11,13] := -0.08345811;
   R_g[11,14] := -0.3010131;
   R_g[11,15] := -0.3438835;
   R_g[12,0] := 0.1546433;
   R_g[12,1] := -0.1955362;
   R_g[12,2] := 0.2216086;
   R_g[12,3] := 0.3276492;
   R_g[12,4] := 0.02648578;
   R_g[12,5] := 0.09656581;
   R_g[12,6] := 0.09269863;
   R_g[12,7] := -0.00748462;
   R_g[12,8] := 0.2384084;
   R_g[12,9] := -0.2226923;
   R_g[12,10] := -0.1432746;
   R_g[12,11] := 0.1678383;
   R_g[12,12] := -1.566237;
   R_g[12,13] := -0.1101629;
   R_g[12,14] := 0.1427753;
   R_g[12,15] := 0.4183835;
   R_g[13,0] := 0.08890279;
   R_g[13,1] := -0.1990502;
   R_g[13,2] := -0.01056181;
   R_g[13,3] := 0.2478623;
   R_g[13,4] := 0.07754356;
   R_g[13,5] := 0.1655405;
   R_g[13,6] := 0.2601499;
   R_g[13,7] := 0.09906179;
   R_g[13,8] := -0.00865919;
   R_g[13,9] := -0.3019298;
   R_g[13,10] := -0.02393581;
   R_g[13,11] := -0.07343359;
   R_g[13,12] := -0.1289207;
   R_g[13,13] := -1.642736;
   R_g[13,14] := 0.06043187;
   R_g[13,15] := 0.1288359;
   R_g[14,0] := -0.09330796;
   R_g[14,1] := 0.1997155;
   R_g[14,2] := -0.1660388;
   R_g[14,3] := -0.2476246;
   R_g[14,4] := -0.245462;
   R_g[14,5] := -0.2337237;
   R_g[14,6] := -0.02659419;
   R_g[14,7] := 0.105768;
   R_g[14,8] := -0.0639934;
   R_g[14,9] := 0.2036995;
   R_g[14,10] := 0.02550231;
   R_g[14,11] := -0.1306159;
   R_g[14,12] := 0.01752861;
   R_g[14,13] := -0.1640865;
   R_g[14,14] := -0.9470394;
   R_g[14,15] := -0.04546883;
   R_g[15,0] := 0.06223761;
   R_g[15,1] := 0.2557459;
   R_g[15,2] := -0.1291973;
   R_g[15,3] := -0.2472079;
   R_g[15,4] := -0.0884731;
   R_g[15,5] := 0.09416921;
   R_g[15,6] := 0.137037;
   R_g[15,7] := 0.01633993;
   R_g[15,8] := -0.00774476;
   R_g[15,9] := 0.1420475;
   R_g[15,10] := -0.01668179;
   R_g[15,11] := -0.2429604;
   R_g[15,12] := -0.174738;
   R_g[15,13] := -0.2071896;
   R_g[15,14] := -0.1961332;
   R_g[15,15] := -1.754754;
   R_o[0,0] := 0.2308647;
   R_o[0,1] := -1.334663;
   R_o[0,2] := 0.4042242;
   R_o[0,3] := 1.004969;
   R_o[0,4] := -0.4504767;
   R_o[0,5] := 0.4184249;
   R_o[0,6] := 0.3334054;
   R_o[0,7] := 0.1674809;
   R_o[0,8] := 0.4531534;
   R_o[0,9] := -0.09557626;
   R_o[0,10] := 0.2930945;
   R_o[0,11] := -1.102839;
   R_o[0,12] := -0.6650082;
   R_o[0,13] := -0.1058089;
   R_o[0,14] := 0.2590909;
   R_o[0,15] := 0.3616749;
   R_o[1,0] := 1.002528;
   R_o[1,1] := -1.37036;
   R_o[1,2] := 0.1954388;
   R_o[1,3] := 0.609374;
   R_o[1,4] := -0.589433;
   R_o[1,5] := 0.5858338;
   R_o[1,6] := -0.09563978;
   R_o[1,7] := 0.2172372;
   R_o[1,8] := 0.6389845;
   R_o[1,9] := 0.4626525;
   R_o[1,10] := -0.08759028;
   R_o[1,11] := -0.1091002;
   R_o[1,12] := -0.5695916;
   R_o[1,13] := -0.1903187;
   R_o[1,14] := 0.5208434;
   R_o[1,15] := -0.1904129;
   R_o[2,0] := 0.6292173;
   R_o[2,1] := -1.097194;
   R_o[2,2] := 0.7218018;
   R_o[2,3] := 0.8983966;
   R_o[2,4] := -0.103797;
   R_o[2,5] := 0.04743656;
   R_o[2,6] := 0.2703439;
   R_o[2,7] := -0.02836194;
   R_o[2,8] := 0.2786625;
   R_o[2,9] := -0.2205554;
   R_o[2,10] := 0.02680908;
   R_o[2,11] := -0.5220854;
   R_o[2,12] := 0.08205704;
   R_o[2,13] := -0.7511023;
   R_o[2,14] := 0.4483716;
   R_o[2,15] := 0.1973718;
   R_o[3,0] := 0.07306311;
   R_o[3,1] := -0.4162663;
   R_o[3,2] := 0.06146695;
   R_o[3,3] := -0.138228;
   R_o[3,4] := -0.1853522;
   R_o[3,5] := 0.131848;
   R_o[3,6] := 0.4892341;
   R_o[3,7] := 0.1009455;
   R_o[3,8] := -0.121296;
   R_o[3,9] := 0.1695517;
   R_o[3,10] := 0.1079443;
   R_o[3,11] := -0.4055073;
   R_o[3,12] := -0.01614563;
   R_o[3,13] := -0.00363492;
   R_o[3,14] := 0.3414511;
   R_o[3,15] := -0.3074647;
   R_o[4,0] := 0.4998139;
   R_o[4,1] := -0.4487727;
   R_o[4,2] := 0.02899466;
   R_o[4,3] := 0.2891186;
   R_o[4,4] := -0.5470661;
   R_o[4,5] := 0.4533124;
   R_o[4,6] := 0.312606;
   R_o[4,7] := 0.2159235;
   R_o[4,8] := -0.1822658;
   R_o[4,9] := -0.08202437;
   R_o[4,10] := 0.1989024;
   R_o[4,11] := -0.445997;
   R_o[4,12] := -0.00842409;
   R_o[4,13] := 0.3160509;
   R_o[4,14] := 0.1949186;
   R_o[4,15] := 0.1517705;
   R_o[5,0] := 0.1672285;
   R_o[5,1] := -0.9065105;
   R_o[5,2] := -0.09893818;
   R_o[5,3] := 0.5721238;
   R_o[5,4] := -0.5256089;
   R_o[5,5] := 0.09904512;
   R_o[5,6] := -0.07018632;
   R_o[5,7] := 0.3906378;
   R_o[5,8] := 0.4664879;
   R_o[5,9] := -0.1485893;
   R_o[5,10] := 0.1839706;
   R_o[5,11] := -0.7344642;
   R_o[5,12] := -0.4822762;
   R_o[5,13] := 0.1130776;
   R_o[5,14] := 0.02705877;
   R_o[5,15] := -0.05367837;
   R_o[6,0] := 0.4642389;
   R_o[6,1] := -1.167083;
   R_o[6,2] := -0.0418876;
   R_o[6,3] := 0.3188611;
   R_o[6,4] := -0.09108678;
   R_o[6,5] := -0.06297291;
   R_o[6,6] := 1.53958;
   R_o[6,7] := -0.626138;
   R_o[6,8] := 0.4499038;
   R_o[6,9] := -0.7262865;
   R_o[6,10] := 0.3824556;
   R_o[6,11] := -0.5390584;
   R_o[6,12] := -0.7175185;
   R_o[6,13] := 0.507979;
   R_o[6,14] := -0.323703;
   R_o[6,15] := -0.09905253;
   R_o[7,0] := 0.290577;
   R_o[7,1] := -1.983839;
   R_o[7,2] := 0.1318081;
   R_o[7,3] := 0.9109895;
   R_o[7,4] := -0.1764812;
   R_o[7,5] := 0.8470377;
   R_o[7,6] := 0.3375674;
   R_o[7,7] := 0.4343486;
   R_o[7,8] := 0.6906033;
   R_o[7,9] := 0.2226612;
   R_o[7,10] := 0.2735369;
   R_o[7,11] := -0.7281427;
   R_o[7,12] := -0.4348153;
   R_o[7,13] := 0.07530996;
   R_o[7,14] := 0.07590891;
   R_o[7,15] := 0.5363369;
   R_o[8,0] := 0.1343116;
   R_o[8,1] := -0.8581089;
   R_o[8,2] := 0.02636042;
   R_o[8,3] := 0.8965567;
   R_o[8,4] := -0.581214;
   R_o[8,5] := 0.1658207;
   R_o[8,6] := 0.3920063;
   R_o[8,7] := 0.4881606;
   R_o[8,8] := -0.4026999;
   R_o[8,9] := -0.1249401;
   R_o[8,10] := -0.1852563;
   R_o[8,11] := -0.5821697;
   R_o[8,12] := -0.1722453;
   R_o[8,13] := -0.06991822;
   R_o[8,14] := 0.4439938;
   R_o[8,15] := 0.06420073;
   R_o[9,0] := 0.6580915;
   R_o[9,1] := -0.7430585;
   R_o[9,2] := 0.04991319;
   R_o[9,3] := 0.7297944;
   R_o[9,4] := -0.1207476;
   R_o[9,5] := -0.1241021;
   R_o[9,6] := 0.2097352;
   R_o[9,7] := 0.6113284;
   R_o[9,8] := 0.6428261;
   R_o[9,9] := -1.041695;
   R_o[9,10] := -1.027741;
   R_o[9,11] := -0.495687;
   R_o[9,12] := -0.7742246;
   R_o[9,13] := 0.2770533;
   R_o[9,14] := 0.6336173;
   R_o[9,15] := 0.3683498;
   R_o[10,0] := 0.1762986;
   R_o[10,1] := -0.8176378;
   R_o[10,2] := -0.4000072;
   R_o[10,3] := 0.3808675;
   R_o[10,4] := -0.04421521;
   R_o[10,5] := 0.1071376;
   R_o[10,6] := 0.4433302;
   R_o[10,7] := 0.2518485;
   R_o[10,8] := 0.5572131;
   R_o[10,9] := -0.3107572;
   R_o[10,10] := -0.1752378;
   R_o[10,11] := -0.2952474;
   R_o[10,12] := -0.62745;
   R_o[10,13] := -0.1415673;
   R_o[10,14] := 0.09456541;
   R_o[10,15] := 0.1587598;
   R_o[11,0] := 0.8746227;
   R_o[11,1] := -1.429159;
   R_o[11,2] := 0.0834833;
   R_o[11,3] := 0.933534;
   R_o[11,4] := -0.2869627;
   R_o[11,5] := 0.6774154;
   R_o[11,6] := 0.3818424;
   R_o[11,7] := 0.1403241;
   R_o[11,8] := 0.4373906;
   R_o[11,9] := 0.1458455;
   R_o[11,10] := 0.205338;
   R_o[11,11] := 0.5737337;
   R_o[11,12] := -0.4247441;
   R_o[11,13] := -0.328859;
   R_o[11,14] := 0.05512207;
   R_o[11,15] := 0.2250471;
   R_o[12,0] := -0.108922;
   R_o[12,1] := -0.7505684;
   R_o[12,2] := -0.2105316;
   R_o[12,3] := 0.4515481;
   R_o[12,4] := -0.9350353;
   R_o[12,5] := 0.3601933;
   R_o[12,6] := 0.3502068;
   R_o[12,7] := 0.08578178;
   R_o[12,8] := 0.1122153;
   R_o[12,9] := 0.2149702;
   R_o[12,10] := 0.01753722;
   R_o[12,11] := -0.6130666;
   R_o[12,12] := -0.4341035;
   R_o[12,13] := 0.2972513;
   R_o[12,14] := 0.461785;
   R_o[12,15] := 0.1768571;
   R_o[13,0] := 0.8438683;
   R_o[13,1] := -0.804963;
   R_o[13,2] := 0.07475836;
   R_o[13,3] := 0.5148878;
   R_o[13,4] := -0.6675235;
   R_o[13,5] := 0.3265819;
   R_o[13,6] := 0.871582;
   R_o[13,7] := -0.14369;
   R_o[13,8] := 0.2130966;
   R_o[13,9] := -0.3292432;
   R_o[13,10] := 0.3362244;
   R_o[13,11] := -0.789337;
   R_o[13,12] := -0.5644252;
   R_o[13,13] := 0.2491675;
   R_o[13,14] := 0.1638097;
   R_o[13,15] := 0.7674901;
   R_o[14,0] := 0.1315343;
   R_o[14,1] := -0.7742588;
   R_o[14,2] := -0.233584;
   R_o[14,3] := 0.6857421;
   R_o[14,4] := -0.4811993;
   R_o[14,5] := -0.2640833;
   R_o[14,6] := 0.5416964;
   R_o[14,7] := -0.191322;
   R_o[14,8] := 0.3080356;
   R_o[14,9] := 0.2251561;
   R_o[14,10] := -0.1517611;
   R_o[14,11] := -0.1808207;
   R_o[14,12] := -0.539659;
   R_o[14,13] := 0.2811023;
   R_o[14,14] := 0.4879507;
   R_o[14,15] := 0.05904227;
   R_o[15,0] := 0.3220614;
   R_o[15,1] := -0.5911628;
   R_o[15,2] := 0.07525509;
   R_o[15,3] := 0.4330951;
   R_o[15,4] := -0.2145242;
   R_o[15,5] := -0.1183812;
   R_o[15,6] := 0.4617145;
   R_o[15,7] := 0.1013162;
   R_o[15,8] := 0.01249216;
   R_o[15,9] := -0.04199028;
   R_o[15,10] := 0.2704256;
   R_o[15,11] := 0.1006244;
   R_o[15,12] := -0.384778;
   R_o[15,13] := -0.120112;
   R_o[15,14] := 0.3695851;
   R_o[15,15] := 0.6734249;
   B_i[0] := 1.39582;
   B_i[1] := 0.6825098;
   B_i[2] := 1.202625;
   B_i[3] := 0.2674634;
   B_i[4] := 1.104314;
   B_i[5] := 0.9527091;
   B_i[6] := 1.367364;
   B_i[7] := 1.247113;
   B_i[8] := 1.512643;
   B_i[9] := 0.1620657;
   B_i[10] := 1.609504;
   B_i[11] := 0.8216099;
   B_i[12] := 1.235464;
   B_i[13] := 1.08166;
   B_i[14] := 0.124677;
   B_i[15] := 0.5498633;
   B_f[0] := 0.7917457;
   B_f[1] := -0.6413339;
   B_f[2] := 1.204501;
   B_f[3] := -1.039677;
   B_f[4] := 1.241214;
   B_f[5] := 0.9316998;
   B_f[6] := 0.5651777;
   B_f[7] := 1.145142;
   B_f[8] := 1.61746;
   B_f[9] := 0.6536825;
   B_f[10] := 0.9096788;
   B_f[11] := -0.5673971;
   B_f[12] := 0.8012313;
   B_f[13] := 0.912231;
   B_f[14] := -1.038805;
   B_f[15] := 1.312093;
   B_g[0] := 0.06687933;
   B_g[1] := -0.683975;
   B_g[2] := 0.5813925;
   B_g[3] := 0.3810755;
   B_g[4] := -0.2204027;
   B_g[5] := 0.3485461;
   B_g[6] := 0.3534212;
   B_g[7] := 0.09094166;
   B_g[8] := -0.1934021;
   B_g[9] := -0.2283598;
   B_g[10] := 0.00825962;
   B_g[11] := 0.1600648;
   B_g[12] := -0.3645913;
   B_g[13] := -0.06400946;
   B_g[14] := 0.2746913;
   B_g[15] := 0.1108486;
   B_o[0] := 2.830544;
   B_o[1] := 2.382227;
   B_o[2] := 2.632618;
   B_o[3] := 1.958189;
   B_o[4] := 2.315962;
   B_o[5] := 2.642084;
   B_o[6] := 3.446781;
   B_o[7] := 3.712433;
   B_o[8] := 2.57036;
   B_o[9] := 2.552044;
   B_o[10] := 2.076454;
   B_o[11] := 2.168941;
   B_o[12] := 2.772432;
   B_o[13] := 3.076823;
   B_o[14] := 1.657935;
   B_o[15] := 2.285517;
   FC_W[0,0] := -0.5330263;
   FC_W[0,1] := 0.682957;
   FC_W[0,2] := -0.6259958;
   FC_W[0,3] := -0.3272032;
   FC_W[0,4] := -0.08957181;
   FC_W[0,5] := -0.1655545;
   FC_W[0,6] := 0.06407359;
   FC_W[0,7] := 0.202257;
   FC_W[0,8] := -1.0473;
   FC_W[0,9] := -1.63025;
   FC_W[0,10] := -0.3651182;
   FC_W[0,11] := -0.6175694;
   FC_W[0,12] := -0.2609785;
   FC_W[0,13] := 0.7963088;
   FC_W[0,14] := 0.06587959;
   FC_W[0,15] := 1.5005;
   FC_W[1,0] := -0.115882;
   FC_W[1,1] := 0.6019747;
   FC_W[1,2] := 0.9843809;
   FC_W[1,3] := -0.1210609;
   FC_W[1,4] := 0.3637234;
   FC_W[1,5] := 0.08963854;
   FC_W[1,6] := -1.693555;
   FC_W[1,7] := -0.8412876;
   FC_W[1,8] := -0.09554562;
   FC_W[1,9] := -0.3392726;
   FC_W[1,10] := 1.170805;
   FC_W[1,11] := 1.692487;
   FC_W[1,12] := -0.02792989;
   FC_W[1,13] := 0.2526466;
   FC_W[1,14] := 1.545473;
   FC_W[1,15] := -0.5985584;
   FC_W[2,0] := -0.5637518;
   FC_W[2,1] := 0.7300333;
   FC_W[2,2] := -0.5408776;
   FC_W[2,3] := -0.4260783;
   FC_W[2,4] := -0.1416197;
   FC_W[2,5] := -0.13633;
   FC_W[2,6] := -0.02574298;
   FC_W[2,7] := 0.2482725;
   FC_W[2,8] := -1.099778;
   FC_W[2,9] := -1.698006;
   FC_W[2,10] := -0.4148934;
   FC_W[2,11] := -0.6640356;
   FC_W[2,12] := -0.2534823;
   FC_W[2,13] := 0.845851;
   FC_W[2,14] := 0.03002551;
   FC_W[2,15] := 1.514569;
   FC_W[3,0] := -0.1913025;
   FC_W[3,1] := 0.2297892;
   FC_W[3,2] := 0.3229723;
   FC_W[3,3] := 0.2144147;
   FC_W[3,4] := 0.316296;
   FC_W[3,5] := -0.00644177;
   FC_W[3,6] := 0.5739819;
   FC_W[3,7] := -0.09706475;
   FC_W[3,8] := -0.05950126;
   FC_W[3,9] := -1.09413;
   FC_W[3,10] := 0.2570405;
   FC_W[3,11] := 0.6612412;
   FC_W[3,12] := -0.3190681;
   FC_W[3,13] := 0.5371132;
   FC_W[3,14] := -1.58714;
   FC_W[3,15] := 0.01048408;
   FC_W[4,0] := 0.3141466;
   FC_W[4,1] := -0.3433263;
   FC_W[4,2] := 0.8911735;
   FC_W[4,3] := -0.7150986;
   FC_W[4,4] := 0.09996962;
   FC_W[4,5] := -0.02766594;
   FC_W[4,6] := 0.512578;
   FC_W[4,7] := -0.9175332;
   FC_W[4,8] := 1.089048;
   FC_W[4,9] := -0.05996554;
   FC_W[4,10] := -1.127543;
   FC_W[4,11] := -0.1694988;
   FC_W[4,12] := -0.7693791;
   FC_W[4,13] := -1.228351;
   FC_W[4,14] := -0.3830509;
   FC_W[4,15] := 1.158476;
   FC_W[5,0] := 0.6665495;
   FC_W[5,1] := -0.5538939;
   FC_W[5,2] := -1.282928;
   FC_W[5,3] := 0.230869;
   FC_W[5,4] := -0.4650589;
   FC_W[5,5] := -2.091754;
   FC_W[5,6] := -0.9611348;
   FC_W[5,7] := 1.042187;
   FC_W[5,8] := 1.518522;
   FC_W[5,9] := -3.803936;
   FC_W[5,10] := -1.478683;
   FC_W[5,11] := -0.2562669;
   FC_W[5,12] := 0.2438862;
   FC_W[5,13] := 0.1155114;
   FC_W[5,14] := -0.3664193;
   FC_W[5,15] := -1.084983;
   FC_W[6,0] := 0.4383626;
   FC_W[6,1] := 0.8904867;
   FC_W[6,2] := 0.1160313;
   FC_W[6,3] := 0.9692903;
   FC_W[6,4] := 1.085123;
   FC_W[6,5] := -0.510233;
   FC_W[6,6] := -0.4337154;
   FC_W[6,7] := 1.296865;
   FC_W[6,8] := -0.1080953;
   FC_W[6,9] := -0.04550074;
   FC_W[6,10] := -0.7336516;
   FC_W[6,11] := 0.2972921;
   FC_W[6,12] := -0.4115362;
   FC_W[6,13] := -0.01893469;
   FC_W[6,14] := -0.8390495;
   FC_W[6,15] := -0.2460979;
   FC_W[7,0] := -0.1847777;
   FC_W[7,1] := 0.2036924;
   FC_W[7,2] := 0.2827305;
   FC_W[7,3] := 0.2577677;
   FC_W[7,4] := 0.3391545;
   FC_W[7,5] := -0.02453313;
   FC_W[7,6] := 0.6303813;
   FC_W[7,7] := -0.0868469;
   FC_W[7,8] := -0.03923411;
   FC_W[7,9] := -1.062993;
   FC_W[7,10] := 0.2598891;
   FC_W[7,11] := 0.6473021;
   FC_W[7,12] := -0.3363241;
   FC_W[7,13] := 0.5315282;
   FC_W[7,14] := -1.569682;
   FC_W[7,15] := 0.01425198;
   FC_W[8,0] := -0.2128507;
   FC_W[8,1] := 0.287179;
   FC_W[8,2] := 0.317035;
   FC_W[8,3] := 0.1540007;
   FC_W[8,4] := 0.3354281;
   FC_W[8,5] := -0.01905481;
   FC_W[8,6] := 0.5331562;
   FC_W[8,7] := -0.09981918;
   FC_W[8,8] := -0.08895166;
   FC_W[8,9] := -1.126273;
   FC_W[8,10] := 0.2581049;
   FC_W[8,11] := 0.6737793;
   FC_W[8,12] := -0.261289;
   FC_W[8,13] := 0.541033;
   FC_W[8,14] := -1.606916;
   FC_W[8,15] := -0.01362194;
   FC_W[9,0] := -0.1954301;
   FC_W[9,1] := 0.2130431;
   FC_W[9,2] := 0.292702;
   FC_W[9,3] := 0.2306473;
   FC_W[9,4] := 0.3276762;
   FC_W[9,5] := -0.02455352;
   FC_W[9,6] := 0.5984318;
   FC_W[9,7] := -0.08202294;
   FC_W[9,8] := -0.06203229;
   FC_W[9,9] := -1.090275;
   FC_W[9,10] := 0.2696502;
   FC_W[9,11] := 0.6541253;
   FC_W[9,12] := -0.3329587;
   FC_W[9,13] := 0.5447234;
   FC_W[9,14] := -1.582466;
   FC_W[9,15] := 0.00871467;
   FC_W[10,0] := -0.4487735;
   FC_W[10,1] := -0.2787283;
   FC_W[10,2] := -0.2087227;
   FC_W[10,3] := -0.5995144;
   FC_W[10,4] := -0.646116;
   FC_W[10,5] := -0.5524399;
   FC_W[10,6] := 0.247803;
   FC_W[10,7] := -0.7400737;
   FC_W[10,8] := 0.3234173;
   FC_W[10,9] := -2.577077;
   FC_W[10,10] := 0.5749816;
   FC_W[10,11] := 0.6185442;
   FC_W[10,12] := 0.01876899;
   FC_W[10,13] := 0.7563331;
   FC_W[10,14] := -0.8973056;
   FC_W[10,15] := -0.3978796;
   FC_W[11,0] := 0.6146721;
   FC_W[11,1] := 0.1916842;
   FC_W[11,2] := 0.9344383;
   FC_W[11,3] := -0.5930158;
   FC_W[11,4] := -0.9233059;
   FC_W[11,5] := 0.4024804;
   FC_W[11,6] := 0.6360304;
   FC_W[11,7] := 0.389712;
   FC_W[11,8] := -0.5143566;
   FC_W[11,9] := -0.2550746;
   FC_W[11,10] := -0.5835565;
   FC_W[11,11] := 0.01116155;
   FC_W[11,12] := -1.250483;
   FC_W[11,13] := -0.2936021;
   FC_W[11,14] := 0.3336428;
   FC_W[11,15] := -1.040676;
   FC_W[12,0] := 0.2221203;
   FC_W[12,1] := -0.1419773;
   FC_W[12,2] := 1.131704;
   FC_W[12,3] := -0.6137382;
   FC_W[12,4] := -0.7516223;
   FC_W[12,5] := 0.4527787;
   FC_W[12,6] := 0.4370326;
   FC_W[12,7] := 0.6888357;
   FC_W[12,8] := -0.2711489;
   FC_W[12,9] := -0.3324692;
   FC_W[12,10] := -0.3672298;
   FC_W[12,11] := -0.2122664;
   FC_W[12,12] := -1.381353;
   FC_W[12,13] := -0.2839057;
   FC_W[12,14] := 0.2129227;
   FC_W[12,15] := -1.02847;
   FC_W[13,0] := -0.4278456;
   FC_W[13,1] := -1.55966;
   FC_W[13,2] := -0.2381402;
   FC_W[13,3] := 0.8133253;
   FC_W[13,4] := 1.017868;
   FC_W[13,5] := -0.7635065;
   FC_W[13,6] := 0.04761689;
   FC_W[13,7] := -0.5287133;
   FC_W[13,8] := -0.08105175;
   FC_W[13,9] := -0.5556808;
   FC_W[13,10] := 1.004662;
   FC_W[13,11] := 1.324528;
   FC_W[13,12] := -1.167233;
   FC_W[13,13] := 1.34941;
   FC_W[13,14] := 2.638295;
   FC_W[13,15] := -0.2266168;
   FC_W[14,0] := -2.358538;
   FC_W[14,1] := 0.4289707;
   FC_W[14,2] := -1.656325;
   FC_W[14,3] := -1.45689;
   FC_W[14,4] := -0.2370753;
   FC_W[14,5] := 2.006904;
   FC_W[14,6] := 1.074223;
   FC_W[14,7] := 2.124806;
   FC_W[14,8] := 1.786735;
   FC_W[14,9] := 0.1440235;
   FC_W[14,10] := -1.981618;
   FC_W[14,11] := 2.800448;
   FC_W[14,12] := 0.03338763;
   FC_W[14,13] := 0.4124092;
   FC_W[14,14] := 1.219082;
   FC_W[14,15] := 0.1871507;
   FC_W[15,0] := 0.9474449;
   FC_W[15,1] := 0.5609007;
   FC_W[15,2] := 0.7729257;
   FC_W[15,3] := -0.4733862;
   FC_W[15,4] := -1.325213;
   FC_W[15,5] := 0.1625959;
   FC_W[15,6] := 0.5493469;
   FC_W[15,7] := -0.0091592;
   FC_W[15,8] := -0.7190735;
   FC_W[15,9] := -0.03908357;
   FC_W[15,10] := -0.9859113;
   FC_W[15,11] := 0.3031035;
   FC_W[15,12] := -0.9841324;
   FC_W[15,13] := 0.09539948;
   FC_W[15,14] := 0.4549902;
   FC_W[15,15] := -0.953172;
   FC_W[16,0] := -0.9079186;
   FC_W[16,1] := 1.470155;
   FC_W[16,2] := 1.468043;
   FC_W[16,3] := -0.3912291;
   FC_W[16,4] := -2.342238;
   FC_W[16,5] := -2.319659;
   FC_W[16,6] := -0.7838322;
   FC_W[16,7] := 0.00836219;
   FC_W[16,8] := 1.982107;
   FC_W[16,9] := 1.165556;
   FC_W[16,10] := -1.210752;
   FC_W[16,11] := 0.5930068;
   FC_W[16,12] := 0.6177696;
   FC_W[16,13] := 3.994448;
   FC_W[16,14] := 0.01262518;
   FC_W[16,15] := 1.049203;
   FC_W[17,0] := -2.798706;
   FC_W[17,1] := -1.420334;
   FC_W[17,2] := 1.690652;
   FC_W[17,3] := -0.668397;
   FC_W[17,4] := 1.273519;
   FC_W[17,5] := 0.02801782;
   FC_W[17,6] := -0.3379328;
   FC_W[17,7] := 2.326567;
   FC_W[17,8] := 2.14158;
   FC_W[17,9] := -0.6385995;
   FC_W[17,10] := 1.597674;
   FC_W[17,11] := -2.156926;
   FC_W[17,12] := -0.7449435;
   FC_W[17,13] := 0.1439934;
   FC_W[17,14] := -0.3848662;
   FC_W[17,15] := 0.08045793;
   FC_W[18,0] := 1.341547;
   FC_W[18,1] := 3.197891;
   FC_W[18,2] := -1.122636;
   FC_W[18,3] := -0.7237122;
   FC_W[18,4] := -1.438901;
   FC_W[18,5] := 1.354497;
   FC_W[18,6] := 1.00367;
   FC_W[18,7] := 0.1155748;
   FC_W[18,8] := 1.428454;
   FC_W[18,9] := -0.04815372;
   FC_W[18,10] := 1.829351;
   FC_W[18,11] := -1.335034;
   FC_W[18,12] := -5.117655;
   FC_W[18,13] := -1.060498;
   FC_W[18,14] := -0.815169;
   FC_W[18,15] := 0.03152023;
   FC_W[19,0] := -0.1523523;
   FC_W[19,1] := -1.047478;
   FC_W[19,2] := 1.241903;
   FC_W[19,3] := -0.4105383;
   FC_W[19,4] := -0.2676516;
   FC_W[19,5] := 0.3593125;
   FC_W[19,6] := 0.1190657;
   FC_W[19,7] := 0.746382;
   FC_W[19,8] := -0.6162935;
   FC_W[19,9] := -0.3676264;
   FC_W[19,10] := -0.647616;
   FC_W[19,11] := -0.01234968;
   FC_W[19,12] := -0.3946634;
   FC_W[19,13] := -0.3151136;
   FC_W[19,14] := 0.3082327;
   FC_W[19,15] := -1.082344;
   FC_W[20,0] := 0.2644098;
   FC_W[20,1] := -1.478355;
   FC_W[20,2] := 0.1183948;
   FC_W[20,3] := -1.160438;
   FC_W[20,4] := -1.161433;
   FC_W[20,5] := 0.02869733;
   FC_W[20,6] := 0.7386208;
   FC_W[20,7] := -0.6949831;
   FC_W[20,8] := 0.4019015;
   FC_W[20,9] := -0.1653061;
   FC_W[20,10] := 0.8912629;
   FC_W[20,11] := 0.3405429;
   FC_W[20,12] := -0.2611554;
   FC_W[20,13] := -0.3854045;
   FC_W[20,14] := 0.6878216;
   FC_W[20,15] := 0.643799;
   FC_W[21,0] := -0.6634615;
   FC_W[21,1] := 0.5873222;
   FC_W[21,2] := 0.06739193;
   FC_W[21,3] := 0.9726313;
   FC_W[21,4] := -0.8678127;
   FC_W[21,5] := -1.02743;
   FC_W[21,6] := 0.1688717;
   FC_W[21,7] := 1.696803;
   FC_W[21,8] := -1.144093;
   FC_W[21,9] := 0.1494212;
   FC_W[21,10] := 0.3269328;
   FC_W[21,11] := 0.6110576;
   FC_W[21,12] := 0.1623239;
   FC_W[21,13] := -1.267441;
   FC_W[21,14] := -0.8775544;
   FC_W[21,15] := 0.542785;
   FC_W[22,0] := 0.2852592;
   FC_W[22,1] := -1.509269;
   FC_W[22,2] := 1.539921;
   FC_W[22,3] := 1.627035;
   FC_W[22,4] := -0.2040465;
   FC_W[22,5] := 0.4312818;
   FC_W[22,6] := -0.04736441;
   FC_W[22,7] := 0.1894242;
   FC_W[22,8] := 0.2640792;
   FC_W[22,9] := -0.9551315;
   FC_W[22,10] := -0.04719095;
   FC_W[22,11] := 1.317374;
   FC_W[22,12] := -0.5620629;
   FC_W[22,13] := -0.3449878;
   FC_W[22,14] := 1.283374;
   FC_W[22,15] := 1.787481;
   FC_W[23,0] := -0.06120704;
   FC_W[23,1] := -1.640421;
   FC_W[23,2] := -0.2532656;
   FC_W[23,3] := 1.119536;
   FC_W[23,4] := 1.086797;
   FC_W[23,5] := -0.3869813;
   FC_W[23,6] := 0.4449602;
   FC_W[23,7] := -0.7841725;
   FC_W[23,8] := 0.07545953;
   FC_W[23,9] := -0.6881379;
   FC_W[23,10] := 0.9839935;
   FC_W[23,11] := 1.540284;
   FC_W[23,12] := -1.133447;
   FC_W[23,13] := 1.854249;
   FC_W[23,14] := 2.036269;
   FC_W[23,15] := -0.3045724;
   FC_W[24,0] := 0.2287794;
   FC_W[24,1] := -1.473234;
   FC_W[24,2] := 1.462772;
   FC_W[24,3] := 1.7643;
   FC_W[24,4] := -0.2494005;
   FC_W[24,5] := 0.4305913;
   FC_W[24,6] := 0.07592186;
   FC_W[24,7] := 0.1482155;
   FC_W[24,8] := 0.3464515;
   FC_W[24,9] := -0.8701573;
   FC_W[24,10] := -0.04559883;
   FC_W[24,11] := 1.239066;
   FC_W[24,12] := -0.7111742;
   FC_W[24,13] := -0.4132386;
   FC_W[24,14] := 1.306507;
   FC_W[24,15] := 1.713007;
   FC_W[25,0] := 0.2286133;
   FC_W[25,1] := -1.475451;
   FC_W[25,2] := 1.462352;
   FC_W[25,3] := 1.765566;
   FC_W[25,4] := -0.2490843;
   FC_W[25,5] := 0.4304071;
   FC_W[25,6] := 0.07507181;
   FC_W[25,7] := 0.1474034;
   FC_W[25,8] := 0.3456639;
   FC_W[25,9] := -0.8683374;
   FC_W[25,10] := -0.04680423;
   FC_W[25,11] := 1.236513;
   FC_W[25,12] := -0.7084648;
   FC_W[25,13] := -0.4137481;
   FC_W[25,14] := 1.304415;
   FC_W[25,15] := 1.71273;
   FC_W[26,0] := 0.3830498;
   FC_W[26,1] := -1.764691;
   FC_W[26,2] := 1.272604;
   FC_W[26,3] := 0.6152487;
   FC_W[26,4] := 0.9249774;
   FC_W[26,5] := 0.4026915;
   FC_W[26,6] := -0.5481057;
   FC_W[26,7] := -0.8134701;
   FC_W[26,8] := 0.5203467;
   FC_W[26,9] := -0.9862843;
   FC_W[26,10] := -0.3936579;
   FC_W[26,11] := 1.143418;
   FC_W[26,12] := 0.1377836;
   FC_W[26,13] := 0.9440991;
   FC_W[26,14] := 1.573741;
   FC_W[26,15] := 0.7988325;
   FC_W[27,0] := -1.142804;
   FC_W[27,1] := 0.5930772;
   FC_W[27,2] := -0.2620744;
   FC_W[27,3] := 0.8762653;
   FC_W[27,4] := -0.9365983;
   FC_W[27,5] := -1.498642;
   FC_W[27,6] := 0.4496078;
   FC_W[27,7] := 1.379625;
   FC_W[27,8] := -1.188017;
   FC_W[27,9] := 0.4169841;
   FC_W[27,10] := 0.3420663;
   FC_W[27,11] := 0.5146847;
   FC_W[27,12] := 0.2882722;
   FC_W[27,13] := -1.382937;
   FC_W[27,14] := -1.011159;
   FC_W[27,15] := 0.1247107;
   FC_W[28,0] := 0.04424974;
   FC_W[28,1] := 0.135361;
   FC_W[28,2] := 0.7555974;
   FC_W[28,3] := -0.3579022;
   FC_W[28,4] := 1.360252;
   FC_W[28,5] := -0.88537;
   FC_W[28,6] := -0.00372644;
   FC_W[28,7] := -0.2996951;
   FC_W[28,8] := 0.1903055;
   FC_W[28,9] := -0.01632601;
   FC_W[28,10] := -1.65227;
   FC_W[28,11] := 0.3413977;
   FC_W[28,12] := -0.3493979;
   FC_W[28,13] := -0.5788615;
   FC_W[28,14] := -0.359042;
   FC_W[28,15] := 0.346769;
   FC_W[29,0] := -0.3855314;
   FC_W[29,1] := 1.27834;
   FC_W[29,2] := -1.677434;
   FC_W[29,3] := -1.057885;
   FC_W[29,4] := 0.2280355;
   FC_W[29,5] := -0.1172309;
   FC_W[29,6] := 0.3620466;
   FC_W[29,7] := -0.448419;
   FC_W[29,8] := 0.0353851;
   FC_W[29,9] := 1.203187;
   FC_W[29,10] := -0.2055158;
   FC_W[29,11] := -1.714249;
   FC_W[29,12] := 0.4914513;
   FC_W[29,13] := 0.4093235;
   FC_W[29,14] := -1.017603;
   FC_W[29,15] := -1.910525;
   FC_W[30,0] := 0.2872345;
   FC_W[30,1] := -1.511201;
   FC_W[30,2] := 1.541994;
   FC_W[30,3] := 1.62218;
   FC_W[30,4] := -0.2022987;
   FC_W[30,5] := 0.43359;
   FC_W[30,6] := -0.05039101;
   FC_W[30,7] := 0.1881196;
   FC_W[30,8] := 0.2618744;
   FC_W[30,9] := -0.9578186;
   FC_W[30,10] := -0.04945299;
   FC_W[30,11] := 1.317318;
   FC_W[30,12] := -0.5575845;
   FC_W[30,13] := -0.3435246;
   FC_W[30,14] := 1.28358;
   FC_W[30,15] := 1.789326;
   FC_W[31,0] := 0.333389;
   FC_W[31,1] := -1.511069;
   FC_W[31,2] := 1.567307;
   FC_W[31,3] := 1.551374;
   FC_W[31,4] := -0.1719055;
   FC_W[31,5] := 0.4543321;
   FC_W[31,6] := -0.0939691;
   FC_W[31,7] := 0.2268038;
   FC_W[31,8] := 0.2382226;
   FC_W[31,9] := -0.98215;
   FC_W[31,10] := -0.06985018;
   FC_W[31,11] := 1.324101;
   FC_W[31,12] := -0.4938571;
   FC_W[31,13] := -0.3189731;
   FC_W[31,14] := 1.264621;
   FC_W[31,15] := 1.823022;
   FC_W[32,0] := 0.2292473;
   FC_W[32,1] := -1.467973;
   FC_W[32,2] := 1.565264;
   FC_W[32,3] := 1.587883;
   FC_W[32,4] := -0.2241208;
   FC_W[32,5] := 0.2562834;
   FC_W[32,6] := -0.05829662;
   FC_W[32,7] := 0.2494973;
   FC_W[32,8] := 0.189134;
   FC_W[32,9] := -0.9591407;
   FC_W[32,10] := -0.00602742;
   FC_W[32,11] := 1.444207;
   FC_W[32,12] := -0.5686611;
   FC_W[32,13] := -0.4541892;
   FC_W[32,14] := 1.218562;
   FC_W[32,15] := 1.79086;
   FC_W[33,0] := 0.2711363;
   FC_W[33,1] := -1.449904;
   FC_W[33,2] := 1.678192;
   FC_W[33,3] := 1.381597;
   FC_W[33,4] := -0.1910754;
   FC_W[33,5] := 0.1816871;
   FC_W[33,6] := -0.2181111;
   FC_W[33,7] := 0.3524041;
   FC_W[33,8] := 0.0608653;
   FC_W[33,9] := -1.059223;
   FC_W[33,10] := -0.01789864;
   FC_W[33,11] := 1.573912;
   FC_W[33,12] := -0.3751651;
   FC_W[33,13] := -0.4647232;
   FC_W[33,14] := 1.117605;
   FC_W[33,15] := 1.886582;
   FC_W[34,0] := 0.3226988;
   FC_W[34,1] := -1.435427;
   FC_W[34,2] := 1.661185;
   FC_W[34,3] := 1.391281;
   FC_W[34,4] := -0.2039064;
   FC_W[34,5] := 0.2631321;
   FC_W[34,6] := -0.2031871;
   FC_W[34,7] := 0.3208036;
   FC_W[34,8] := 0.1088318;
   FC_W[34,9] := -1.062686;
   FC_W[34,10] := -0.01133159;
   FC_W[34,11] := 1.513079;
   FC_W[34,12] := -0.4399895;
   FC_W[34,13] := -0.4157502;
   FC_W[34,14] := 1.146734;
   FC_W[34,15] := 1.899761;
   FC_W[35,0] := 0.1840785;
   FC_W[35,1] := -1.462723;
   FC_W[35,2] := 1.473073;
   FC_W[35,3] := 1.667966;
   FC_W[35,4] := -0.2405721;
   FC_W[35,5] := 0.2115589;
   FC_W[35,6] := 0.05332418;
   FC_W[35,7] := 0.2106999;
   FC_W[35,8] := 0.2360089;
   FC_W[35,9] := -0.891493;
   FC_W[35,10] := 0.048077;
   FC_W[35,11] := 1.427772;
   FC_W[35,12] := -0.7111167;
   FC_W[35,13] := -0.4602369;
   FC_W[35,14] := 1.258088;
   FC_W[35,15] := 1.702616;
   FC_W[36,0] := -2.863858;
   FC_W[36,1] := -0.52148;
   FC_W[36,2] := -0.296759;
   FC_W[36,3] := 4.633551;
   FC_W[36,4] := -1.540046;
   FC_W[36,5] := 0.8701387;
   FC_W[36,6] := 1.445184;
   FC_W[36,7] := -2.182616;
   FC_W[36,8] := 0.8216071;
   FC_W[36,9] := -0.1750247;
   FC_W[36,10] := -0.9630795;
   FC_W[36,11] := -1.566791;
   FC_W[36,12] := -0.4161453;
   FC_W[36,13] := -0.6984285;
   FC_W[36,14] := 1.355617;
   FC_W[36,15] := -0.05721238;
   FC_W[37,0] := 0.1548835;
   FC_W[37,1] := -1.455895;
   FC_W[37,2] := 1.444182;
   FC_W[37,3] := 1.711339;
   FC_W[37,4] := -0.2441721;
   FC_W[37,5] := 0.1982007;
   FC_W[37,6] := 0.08134115;
   FC_W[37,7] := 0.1947857;
   FC_W[37,8] := 0.2436527;
   FC_W[37,9] := -0.8714406;
   FC_W[37,10] := 0.05783046;
   FC_W[37,11] := 1.419663;
   FC_W[37,12] := -0.7412031;
   FC_W[37,13] := -0.4580342;
   FC_W[37,14] := 1.272599;
   FC_W[37,15] := 1.667308;
   FC_W[38,0] := -0.2153435;
   FC_W[38,1] := -1.963263;
   FC_W[38,2] := -0.7550882;
   FC_W[38,3] := 1.207781;
   FC_W[38,4] := -1.464495;
   FC_W[38,5] := -0.2194848;
   FC_W[38,6] := -3.290615;
   FC_W[38,7] := -0.7485562;
   FC_W[38,8] := 0.2515741;
   FC_W[38,9] := 1.207716;
   FC_W[38,10] := -0.3075515;
   FC_W[38,11] := 0.9888396;
   FC_W[38,12] := -0.9664539;
   FC_W[38,13] := 1.244482;
   FC_W[38,14] := -2.634727;
   FC_W[38,15] := 1.384281;
   FC_W[39,0] := -1.4608;
   FC_W[39,1] := -0.9021818;
   FC_W[39,2] := -1.388807;
   FC_W[39,3] := -0.08306644;
   FC_W[39,4] := -0.668493;
   FC_W[39,5] := 1.325439;
   FC_W[39,6] := -1.175365;
   FC_W[39,7] := 0.8160962;
   FC_W[39,8] := 1.067329;
   FC_W[39,9] := 0.5814661;
   FC_W[39,10] := -1.257989;
   FC_W[39,11] := 2.078559;
   FC_W[39,12] := -0.3857729;
   FC_W[39,13] := 0.6238445;
   FC_W[39,14] := -0.8135812;
   FC_W[39,15] := 0.8960469;
   FC_B[0] := 0.02629896;
   FC_B[1] := 0.4275232;
   FC_B[2] := 0.01502107;
   FC_B[3] := -0.1018768;
   FC_B[4] := -0.3340568;
   FC_B[5] := 0.4180066;
   FC_B[6] := 0.2690993;
   FC_B[7] := -0.1066804;
   FC_B[8] := -0.05807845;
   FC_B[9] := -0.1029649;
   FC_B[10] := 0.06830941;
   FC_B[11] := -0.8202225;
   FC_B[12] := -0.823633;
   FC_B[13] := -0.4874749;
   FC_B[14] := 0.4063556;
   FC_B[15] := -0.7498074;
   FC_B[16] := 0.5293838;
   FC_B[17] := -0.02519251;
   FC_B[18] := 0.7223178;
   FC_B[19] := -0.9723449;
   FC_B[20] := -0.6660115;
   FC_B[21] := 0.1745601;
   FC_B[22] := -1.324046;
   FC_B[23] := -0.7062744;
   FC_B[24] := -1.307876;
   FC_B[25] := -1.307821;
   FC_B[26] := -1.029755;
   FC_B[27] := 0.4372153;
   FC_B[28] := 0.05014376;
   FC_B[29] := 1.186533;
   FC_B[30] := -1.325034;
   FC_B[31] := -1.32861;
   FC_B[32] := -1.279171;
   FC_B[33] := -1.260758;
   FC_B[34] := -1.279813;
   FC_B[35] := -1.260518;
   FC_B[36] := -0.3418005;
   FC_B[37] := -1.24987;
   FC_B[38] := 0.5024799;
   FC_B[39] := 0.4692824;

END_DATA_BLOCK

FUNCTION "_RestartTesting" : Int
{ S7_Optimized_Access := 'TRUE' }
VERSION : 0.1
   VAR_INPUT
      bStart : Bool;
   END_VAR


BEGIN
	IF #bStart THEN
	    "DB_Main".PredictCount := 0;
	    "DB_Result".TruePositive := 0;
	    "DB_Result".TrueNegative := 0;
	    "DB_Result".FalsePositive := 0;
	    "DB_Result".FalseNegative := 0;
	    #_RestartTesting := 10;
	ELSE
	    #_RestartTesting := 0;
	END_IF;
END_FUNCTION

FUNCTION "_Zscore" : Real
{ S7_Optimized_Access := 'TRUE' }
VERSION : 0.1
   VAR_INPUT
      iRow : Int;
      iCol : Int;
   END_VAR


BEGIN
	#_Zscore := ("DB_Attack_v0_first_attack".DATA[#iRow, #iCol] - "DB_FeatureNormRef_Means".Means[#iCol]) / "DB_FeatureNormRef_std".std[#iCol];

END_FUNCTION

FUNCTION "_LIMIT" : Real
{ S7_Optimized_Access := 'TRUE' }
VERSION : 0.1
   VAR_INPUT
      inVal : Real;
      minVal : Real;
      maxVal : Real;
   END_VAR

   VAR_TEMP
      lo : Real;
      hi : Real;
   END_VAR


BEGIN
	IF #inVal < #minVal THEN
	    #_LIMIT := #minVal;
	ELSIF #inVal > #maxVal THEN
	    #_LIMIT := #maxVal;
	ELSE
	    #_LIMIT := #inVal;
	END_IF;

END_FUNCTION

FUNCTION "_FC_layer" : Void
{ S7_Optimized_Access := 'TRUE' }
VERSION : 0.1
   VAR_INPUT
      h_t : Array[0..15] of Real;
   END_VAR

   VAR_OUTPUT
      y : Array[0..39] of Real;
   END_VAR

   VAR_TEMP
      i : Int;
      j : Int;
   END_VAR


BEGIN
	FOR #i := 0 TO 39 DO
	    #y[#i] := 0.0;
	    FOR #j := 0 TO 15 DO
	        #y[#i] := #y[#i] + "DB_model_HS16_IW100".FC_W[#i, #j] * #h_t[#j];
	    END_FOR;
	    #y[#i] := #y[#i] + "DB_model_HS16_IW100".FC_B[#i];
	END_FOR;
END_FUNCTION

DATA_BLOCK "DB_Measuring"
{ S7_Optimized_Access := 'TRUE' }
VERSION : 0.1
NON_RETAIN
   VAR
      CycleTime_ms : DInt;
      last_cycle_time : LTime;
      last_cycle_ms : Array[0..3000] of DInt;
   END_VAR


BEGIN

END_DATA_BLOCK

DATA_BLOCK "DB_LSTM"
{ S7_Optimized_Access := 'TRUE' }
VERSION : 0.1
NON_RETAIN
   VAR
      c_tm1 : Array[0..15] of Real;
      h_tm1 : Array[0..15] of Real;
      x_t : Array[0..99, 0..39] of Real;
      c_t : Array[0..15] of Real;
      h_t : Array[0..15] of Real;
      y : Array[0..39] of Real;
   END_VAR


BEGIN

END_DATA_BLOCK

ORGANIZATION_BLOCK "Main"
TITLE = "Main Program Sweep (Cycle)"
{ S7_Optimized_Access := 'TRUE' }
VERSION : 0.1
   VAR_TEMP
      f_t : Array[0..15] of Real;
      g_t : Array[0..15] of Real;
      o_t : Array[0..15] of Real;
      x_ct : Real;
      x_o : Real;
      x_g : Real;
      i_t : Array[0..15] of Real;
      x_f : Real;
      x_i : Real;
      k : Int;
      t : Int;
      I : Int;
      j : Int;
      vInfo : Variant;
      lastCycleTime : DInt;
      predicted_class : Int;
      retVal : Int;
   END_VAR


BEGIN
	        //-->> Cycle Time measuring
	#retVal:= RT_INFO(
	                  MODE := 25,
	                  OB := 1,
	                  INFO := "DB_Measuring".last_cycle_time
	);
	"DB_Measuring".last_cycle_ms["DB_Main".PredictCount]:= LTIME_TO_DINT("DB_Measuring".last_cycle_time);
	"DB_Measuring".CycleTime_ms := LTIME_TO_DINT("DB_Measuring".last_cycle_time) /1000000;


	 CASE "DB_Main".iState OF
	        //-->> IDLE
	    0:
	        "DB_Main".iState := "_RestartTesting"("DB_Main".bStart);


	        //-->> Fill Model Window
	    10:
	        FOR #I := 0 TO 15 DO
	            "DB_LSTM".h_tm1[#I] := 0.0;
	            "DB_LSTM".c_tm1[#I] := 0.0;
	        END_FOR;

	        FOR #I := 0 TO 99 DO
	            FOR #j := 0 TO 39 DO
	                "DB_LSTM".x_t[#I, #j] := "_Zscore"(iRow := #I, iCol := #j);
	            END_FOR;
	        END_FOR;
	        "DB_Result".TrueNegative := 100;
	        "DB_Main".PredictCount := 100;
	        "DB_Main".iState := 20;


	        //-->> Call LSTM modell
	    20:
	        FOR #I := 0 TO 15 DO
	            "DB_LSTM".c_tm1[#I] := 0.0;
	            "DB_LSTM".h_tm1[#I] := 0.0;
	        END_FOR;

	        FOR #t := 0 TO 99 DO
	            FOR #I := 0 TO 15 DO

	                // ---- Input gate ----
	                #x_i := "DB_model_HS16_IW100".B_i[#I];
	                FOR #k := 0 TO 39 DO
	                    #x_i := #x_i
	                    + "DB_model_HS16_IW100".W_i[#I, #k]
	                    * "DB_LSTM".x_t[#t, #k];
	                END_FOR;
	                FOR #j := 0 TO 15 DO
	                    #x_i := #x_i
	                    + "DB_model_HS16_IW100".R_i[#I, #j]
	                    * "DB_LSTM".h_tm1[#j];
	                END_FOR;
	                #x_i := "_LIMIT"(inVal := #x_i, maxVal := 20, minVal := -20);
	                #i_t[#I] := 1.0 / (1.0 + EXP(- #x_i));

	                // ---- Forget gate ----
	                #x_f := "DB_model_HS16_IW100".B_f[#I];
	                FOR #k := 0 TO 39 DO
	                    #x_f := #x_f
	                    + "DB_model_HS16_IW100".W_f[#I, #k]
	                    * "DB_LSTM".x_t[#t, #k];
	                END_FOR;
	                FOR #j := 0 TO 15 DO
	                    #x_f := #x_f
	                    + "DB_model_HS16_IW100".R_f[#I, #j]
	                    * "DB_LSTM".h_tm1[#j];
	                END_FOR;
	                #x_f := "_LIMIT"(inVal := #x_f, maxVal := 20, minVal := -20);
	                #f_t[#I] := 1.0 / (1.0 + EXP(- #x_f));

	                // ---- Cell candidate (tanh) ----
	                #x_g := "DB_model_HS16_IW100".B_g[#I];
	                FOR #k := 0 TO 39 DO
	                    #x_g := #x_g
	                    + "DB_model_HS16_IW100".W_g[#I, #k]
	                    * "DB_LSTM".x_t[#t, #k];
	                END_FOR;
	                FOR #j := 0 TO 15 DO
	                    #x_g := #x_g
	                    + "DB_model_HS16_IW100".R_g[#I, #j]
	                    * "DB_LSTM".h_tm1[#j];
	                END_FOR;
	                #x_g := "_LIMIT"(inVal := #x_g, maxVal := 20, minVal := -20);
	                #g_t[#I] := (EXP(#x_g) - EXP(- #x_g)) / (EXP(#x_g) + EXP(- #x_g)); // tanh

	                // ---- Output gate (sigmoid) ----
	                #x_o := "DB_model_HS16_IW100".B_o[#I];
	                FOR #k := 0 TO 39 DO
	                    #x_o := #x_o
	                    + "DB_model_HS16_IW100".W_o[#I, #k]
	                    * "DB_LSTM".x_t[#t, #k];
	                END_FOR;
	                FOR #j := 0 TO 15 DO
	                    #x_o := #x_o
	                    + "DB_model_HS16_IW100".R_o[#I, #j]
	                    * "DB_LSTM".h_tm1[#j];
	                END_FOR;
	                #x_o := "_LIMIT"(inVal := #x_o, maxVal := 20, minVal := -20);
	                #o_t[#I] := 1.0 / (1.0 + EXP(- #x_o));

	                // ---- Cell state update ----
	                "DB_LSTM".c_t[#I] := #f_t[#I] * "DB_LSTM".c_tm1[#I] + #i_t[#I] * #g_t[#I];

	                // ---- Hidden state (tanh) ----
	                #x_ct := "_LIMIT"(inVal := "DB_LSTM".c_t[#I], maxVal := 20, minVal := -20);
	                "DB_LSTM".h_t[#I] := #o_t[#I] * ((EXP(#x_ct) - EXP(- #x_ct)) / (EXP(#x_ct) + EXP(- #x_ct)));
	            END_FOR;


	            FOR #I := 0 TO 15 DO
	                "DB_LSTM".c_tm1[#I] := "DB_LSTM".c_t[#I];
	                "DB_LSTM".h_tm1[#I] := "DB_LSTM".h_t[#I];
	            END_FOR;
	        END_FOR;

	        // Fully connected layer
	        "_FC_layer"(h_t := "DB_LSTM".h_t,
	                    y => "DB_LSTM".y);

	        // MSE
	        "DB_Main".Mse := 0.0;
	        FOR #k := 0 TO 39 DO
	            "DB_Main".Mse := "DB_Main".Mse
	            + ("DB_LSTM".x_t[99, #k] - "DB_LSTM".y[#k])
	            * ("DB_LSTM".x_t[99, #k] - "DB_LSTM".y[#k]);
	        END_FOR;
	        "DB_Main".Mse := "DB_Main".Mse / INT_TO_REAL(40);

	        // Attack / Normal
	        IF "DB_Main".Mse > "DB_Result".THRESHOLD THEN
	            #predicted_class := 1;  // Attack
	        ELSE
	            #predicted_class := 0;  // Normal
	        END_IF;
	        "DB_Result".Predicted_class := #predicted_class;

	        IF "DB_Result".Predicted_class = 1 AND
	            REAL_TO_INT("DB_Attack_v0_first_attack".DATA["DB_Main".PredictCount, 40]) = 1
	        THEN
	            "DB_Result".TruePositive := "DB_Result".TruePositive + 1;
	        ELSIF "DB_Result".Predicted_class = 0 AND
	            REAL_TO_INT("DB_Attack_v0_first_attack".DATA["DB_Main".PredictCount, 40]) = 0
	        THEN
	            "DB_Result".TrueNegative := "DB_Result".TrueNegative + 1;
	        ELSIF "DB_Result".Predicted_class = 1 AND
	            REAL_TO_INT("DB_Attack_v0_first_attack".DATA["DB_Main".PredictCount, 40]) = 0
	        THEN
	            "DB_Result".FalsePositive := "DB_Result".FalsePositive + 1;
	        ELSIF "DB_Result".Predicted_class = 0 AND
	            REAL_TO_INT("DB_Attack_v0_first_attack".DATA["DB_Main".PredictCount, 40]) = 1
	        THEN
	            "DB_Result".FalseNegative := "DB_Result".FalseNegative + 1;
	        END_IF;
	        "DB_Main".PredictCount := "DB_Main".PredictCount + 1;

	        IF "DB_Main".PredictCount >= "DB_Result".EXPECTED_PREDICITON_COUNT THEN
	            "DB_Main".iState := 100;
	        ELSE

	            FOR #I := 0 TO 98 DO
	                FOR #j := 0 TO 39 DO
	                    "DB_LSTM".x_t[#I, #j] := "DB_LSTM".x_t[#I + 1, #j];
	                END_FOR;
	            END_FOR;

	            FOR #j := 0 TO 39 DO
	                "DB_LSTM".x_t[99, #j] := "_Zscore"(iRow := "DB_Main".PredictCount, iCol := #j);
	            END_FOR;
	            "DB_Main".iState := 20;
	        END_IF;


	        //-->> Test Ready Compare Result
	    100:
	        IF "DB_Result".TrueNegative <> "DB_Result".EXPECTED_TRUE_NEGATIVE THEN
	            "DB_Result".MismatchCount := "DB_Result".MismatchCount + 1;
	        END_IF;
	        IF "DB_Result".FalsePositive <>"DB_Result".EXPECTED_FALSE_POSITIVE THEN
	            "DB_Result".MismatchCount := "DB_Result".MismatchCount + 1;
	        END_IF;
	        IF "DB_Result".FalseNegative <> "DB_Result".EXPECTED_FALSE_NEGATIVE THEN
	            "DB_Result".MismatchCount := "DB_Result".MismatchCount + 1;
	        END_IF;
	        IF "DB_Result".TruePositive <> "DB_Result".EXPECTED_TRUE_POSITIVE THEN
	            "DB_Result".MismatchCount := "DB_Result".MismatchCount + 1;
	        END_IF;
	        IF "DB_Main".PredictCount <> "DB_Result".EXPECTED_PREDICITON_COUNT THEN
	            "DB_Result".MismatchCount := "DB_Result".MismatchCount + 1;
	        END_IF;
	        IF "DB_Result".MismatchCount <> 0 THEN
	            "DB_Main".iState := 150;
	        ELSE
	            "DB_Main".iState := 200;
	        END_IF;

	    150,200:
	        IF NOT "DB_Main".bStart THEN
	            "DB_Main".iState := 0;
	        END_IF;

	  END_CASE;
END_ORGANIZATION_BLOCK

